Yaskawa INFORM job: aprem2TRJ0.JBI

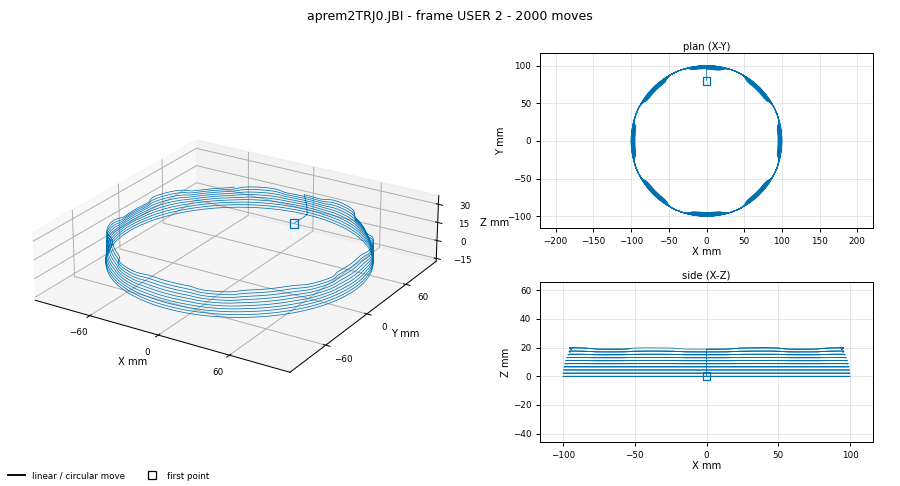
[picture p0: tool path of aprem2TRJ0.JBI in frame USER 2, 2000 of 2000 moves have a stored position in this frame; points joined in program order, loops and branches not executed]
/JOB
//NAME aprem2TRJ0
//POS
///NPOS 2000,0,2000,0,0,0
///USER 2
///TOOL 1
///POSTYPE USER
///RECTAN
///RCONF 1,0,0,0,0,0,0,0,0,0,0,0,0,0,0,0,0,0,0,0,0,0,0,0
C00000=0.000,80.000,0.000,-180.0000,0.0000,0.0000
C00001=0.000,100.000,0.000,-180.0000,0.0000,0.0000
C00002=5.792,99.832,0.000,-180.0000,-0.0000,0.0000
C00003=10.988,99.394,0.000,-180.0000,-0.0000,0.0000
C00004=15.564,98.781,0.000,-180.0000,-0.0000,0.0000
C00005=18.698,98.237,0.000,-180.0000,-0.0000,0.0000
C00006=20.854,97.801,0.000,-180.0000,-0.0000,0.0000
C00007=22.593,97.414,0.000,-180.0000,-0.0000,0.0000
C00008=24.351,96.990,0.000,-180.0000,-0.0000,0.0000
C00009=26.550,96.411,0.000,-180.0000,-0.0000,0.0000
C00010=29.248,95.627,0.000,-180.0000,-0.0000,0.0000
C00011=32.094,94.710,0.000,-180.0000,-0.0000,0.0000
C00012=34.739,93.772,0.000,-180.0000,-0.0000,0.0000
C00013=37.121,92.855,0.000,-180.0000,-0.0000,0.0000
C00014=39.410,91.907,0.000,-180.0000,-0.0000,0.0000
C00015=41.743,90.871,0.000,-180.0000,-0.0000,0.0000
C00016=44.276,89.664,0.000,180.0000,0.0000,0.0000
C00017=46.937,88.300,0.000,180.0000,0.0000,0.0000
C00018=49.400,86.946,0.000,-180.0000,-0.0000,0.0000
C00019=51.363,85.801,0.000,-180.0000,-0.0000,0.0000
C00020=52.906,84.858,0.000,-180.0000,-0.0000,0.0000
C00021=54.410,83.902,0.000,-180.0000,-0.0000,0.0000
C00022=56.242,82.685,0.000,-180.0000,-0.0000,0.0000
C00023=58.844,80.854,0.000,-180.0000,-0.0000,0.0000
C00024=62.512,78.053,0.000,-180.0000,-0.0000,0.0000
C00025=66.496,74.687,0.000,-180.0000,-0.0000,0.0000
C00026=70.711,70.711,0.000,-180.0000,-0.0000,0.0000
C00027=74.687,66.496,0.000,-180.0000,-0.0000,0.0000
C00028=78.053,62.512,0.000,-180.0000,-0.0000,0.0000
C00029=80.854,58.844,0.000,180.0000,0.0000,0.0000
C00030=82.685,56.242,0.000,-180.0000,-0.0000,0.0000
C00031=83.902,54.410,0.000,-180.0000,-0.0000,0.0000
C00032=84.858,52.906,0.000,-180.0000,-0.0000,0.0000
C00033=85.801,51.363,0.000,-180.0000,-0.0000,0.0000
C00034=86.946,49.400,0.000,-180.0000,-0.0000,0.0000
C00035=88.300,46.937,0.000,-180.0000,-0.0000,0.0000
C00036=89.664,44.276,0.000,-180.0000,-0.0000,0.0000
C00037=90.871,41.743,0.000,-180.0000,-0.0000,0.0000
C00038=91.907,39.410,0.000,-180.0000,-0.0000,0.0000
C00039=92.855,37.121,0.000,-180.0000,-0.0000,0.0000
C00040=93.772,34.739,0.000,-180.0000,-0.0000,0.0000
C00041=94.710,32.094,0.000,-180.0000,-0.0000,0.0000
C00042=95.627,29.248,0.000,-180.0000,-0.0000,0.0000
C00043=96.411,26.550,0.000,-180.0000,-0.0000,0.0000
C00044=96.990,24.351,0.000,-180.0000,-0.0000,0.0000
C00045=97.414,22.593,0.000,-180.0000,-0.0000,0.0000
C00046=97.801,20.854,0.000,-180.0000,-0.0000,0.0000
C00047=98.237,18.698,0.000,-180.0000,-0.0000,0.0000
C00048=98.781,15.564,0.000,-180.0000,-0.0000,0.0000
C00049=99.394,10.988,0.000,-180.0000,-0.0000,0.0000
C00050=99.832,5.792,0.000,-180.0000,-0.0000,0.0000
C00051=100.000,0.000,0.000,-180.0000,-0.0000,0.0000
C00052=99.832,-5.792,0.000,180.0000,-0.0000,0.0000
C00053=99.394,-10.988,0.000,180.0000,-0.0000,0.0000
C00054=98.781,-15.564,0.000,180.0000,-0.0000,0.0000
C00055=98.237,-18.698,0.000,180.0000,-0.0000,0.0000
C00056=97.801,-20.854,0.000,180.0000,-0.0000,0.0000
C00057=97.414,-22.593,0.000,180.0000,-0.0000,0.0000
C00058=96.990,-24.351,0.000,180.0000,-0.0000,0.0000
C00059=96.411,-26.550,0.000,180.0000,-0.0000,0.0000
C00060=95.627,-29.248,0.000,180.0000,-0.0000,0.0000
C00061=94.710,-32.094,0.000,180.0000,-0.0000,0.0000
C00062=93.772,-34.739,0.000,180.0000,-0.0000,0.0000
C00063=92.855,-37.121,0.000,180.0000,-0.0000,0.0000
C00064=91.907,-39.410,0.000,180.0000,-0.0000,0.0000
C00065=90.871,-41.743,0.000,180.0000,-0.0000,0.0000
C00066=89.664,-44.276,0.000,180.0000,-0.0000,0.0000
C00067=88.300,-46.937,0.000,180.0000,-0.0000,0.0000
C00068=86.946,-49.400,0.000,180.0000,-0.0000,0.0000
C00069=85.801,-51.363,0.000,180.0000,-0.0000,0.0000
C00070=84.858,-52.906,0.000,180.0000,-0.0000,0.0000
C00071=83.902,-54.410,0.000,180.0000,-0.0000,0.0000
C00072=82.685,-56.242,0.000,180.0000,-0.0000,0.0000
C00073=80.854,-58.844,0.000,180.0000,-0.0000,0.0000
C00074=78.053,-62.512,0.000,180.0000,-0.0000,0.0000
C00075=74.687,-66.496,0.000,180.0000,-0.0000,0.0000
C00076=70.711,-70.711,0.000,180.0000,-0.0000,0.0000
C00077=66.496,-74.687,0.000,180.0000,-0.0000,0.0000
C00078=62.512,-78.053,0.000,180.0000,-0.0000,0.0000
C00079=58.844,-80.854,0.000,180.0000,-0.0000,0.0000
C00080=56.242,-82.685,0.000,180.0000,-0.0000,0.0000
C00081=54.410,-83.902,0.000,180.0000,-0.0000,0.0000
C00082=52.906,-84.858,0.000,180.0000,-0.0000,0.0000
C00083=51.363,-85.801,0.000,180.0000,-0.0000,0.0000
C00084=49.400,-86.946,0.000,-180.0000,0.0000,0.0000
C00085=46.937,-88.300,0.000,180.0000,-0.0000,0.0000
C00086=44.276,-89.664,0.000,180.0000,-0.0000,0.0000
C00087=41.743,-90.871,0.000,180.0000,-0.0000,0.0000
C00088=39.410,-91.907,0.000,180.0000,-0.0000,0.0000
C00089=37.121,-92.855,0.000,180.0000,-0.0000,0.0000
C00090=34.739,-93.772,0.000,180.0000,-0.0000,0.0000
C00091=32.094,-94.710,0.000,180.0000,-0.0000,0.0000
C00092=29.248,-95.627,0.000,180.0000,-0.0000,0.0000
C00093=26.550,-96.411,0.000,180.0000,-0.0000,0.0000
C00094=24.351,-96.990,0.000,180.0000,-0.0000,0.0000
C00095=22.593,-97.414,0.000,180.0000,-0.0000,0.0000
C00096=20.854,-97.801,0.000,180.0000,-0.0000,0.0000
C00097=18.698,-98.237,0.000,180.0000,-0.0000,0.0000
C00098=15.564,-98.781,0.000,180.0000,-0.0000,0.0000
C00099=10.988,-99.394,0.000,180.0000,-0.0000,0.0000
C00100=5.792,-99.832,0.000,180.0000,-0.0000,0.0000
C00101=0.000,-100.000,0.000,-180.0000,-0.0000,0.0000
C00102=0.000,-100.000,0.000,-180.0000,-0.0000,0.0000
C00103=-5.792,-99.832,0.000,-180.0000,-0.0000,0.0000
C00104=-10.988,-99.394,0.000,-180.0000,-0.0000,0.0000
C00105=-15.564,-98.781,0.000,-180.0000,-0.0000,0.0000
C00106=-18.698,-98.237,0.000,-180.0000,-0.0000,0.0000
C00107=-20.854,-97.801,0.000,-180.0000,-0.0000,0.0000
C00108=-22.593,-97.414,0.000,-180.0000,-0.0000,0.0000
C00109=-24.351,-96.990,0.000,-180.0000,-0.0000,0.0000
C00110=-26.550,-96.411,0.000,-180.0000,-0.0000,0.0000
C00111=-29.248,-95.627,0.000,-180.0000,-0.0000,0.0000
C00112=-32.094,-94.710,0.000,-180.0000,-0.0000,0.0000
C00113=-34.739,-93.772,0.000,-180.0000,-0.0000,0.0000
C00114=-37.121,-92.855,0.000,-180.0000,-0.0000,0.0000
C00115=-39.410,-91.907,0.000,-180.0000,-0.0000,0.0000
C00116=-41.743,-90.871,0.000,-180.0000,-0.0000,0.0000
C00117=-44.276,-89.664,0.000,-180.0000,-0.0000,0.0000
C00118=-46.937,-88.300,0.000,-180.0000,-0.0000,0.0000
C00119=-49.400,-86.946,0.000,-180.0000,-0.0000,0.0000
C00120=-51.363,-85.801,0.000,-180.0000,-0.0000,0.0000
C00121=-52.906,-84.858,0.000,-180.0000,-0.0000,0.0000
C00122=-54.410,-83.902,0.000,-180.0000,-0.0000,0.0000
C00123=-56.242,-82.685,0.000,-180.0000,-0.0000,0.0000
C00124=-58.844,-80.854,0.000,-180.0000,-0.0000,0.0000
C00125=-62.512,-78.053,0.000,-180.0000,-0.0000,0.0000
C00126=-66.496,-74.687,0.000,-180.0000,-0.0000,0.0000
C00127=-70.711,-70.711,0.000,-180.0000,-0.0000,0.0000
C00128=-74.687,-66.496,0.000,-180.0000,-0.0000,0.0000
C00129=-78.053,-62.512,0.000,-180.0000,-0.0000,0.0000
C00130=-80.854,-58.844,0.000,-180.0000,-0.0000,0.0000
C00131=-82.685,-56.242,0.000,-180.0000,-0.0000,0.0000
C00132=-83.902,-54.410,0.000,-180.0000,-0.0000,0.0000
C00133=-84.858,-52.906,0.000,-180.0000,-0.0000,0.0000
C00134=-85.801,-51.363,0.000,-180.0000,-0.0000,0.0000
C00135=-86.946,-49.400,0.000,-180.0000,-0.0000,0.0000
C00136=-88.300,-46.937,0.000,-180.0000,-0.0000,0.0000
C00137=-89.664,-44.276,0.000,-180.0000,-0.0000,0.0000
C00138=-90.871,-41.743,0.000,180.0000,0.0000,0.0000
C00139=-91.907,-39.410,0.000,180.0000,0.0000,0.0000
C00140=-92.855,-37.121,0.000,-180.0000,-0.0000,0.0000
C00141=-93.772,-34.739,0.000,-180.0000,-0.0000,0.0000
C00142=-94.710,-32.094,0.000,180.0000,0.0000,0.0000
C00143=-95.627,-29.248,0.000,180.0000,0.0000,0.0000
C00144=-96.411,-26.550,0.000,-180.0000,-0.0000,0.0000
C00145=-96.990,-24.351,0.000,-180.0000,-0.0000,0.0000
C00146=-97.414,-22.593,0.000,-180.0000,-0.0000,0.0000
C00147=-97.801,-20.854,0.000,-180.0000,-0.0000,0.0000
C00148=-98.237,-18.698,0.000,-180.0000,-0.0000,0.0000
C00149=-98.781,-15.564,0.000,-180.0000,-0.0000,0.0000
C00150=-99.394,-10.988,0.000,-180.0000,-0.0000,0.0000
C00151=-99.832,-5.792,0.000,-180.0000,-0.0000,0.0000
C00152=-100.000,0.000,0.000,180.0000,0.0000,0.0000
C00153=-99.832,5.792,0.000,-180.0000,0.0000,0.0000
C00154=-99.394,10.988,0.000,-180.0000,0.0000,0.0000
C00155=-98.781,15.564,0.000,-180.0000,0.0000,0.0000
C00156=-98.237,18.698,0.000,-180.0000,0.0000,0.0000
C00157=-97.801,20.854,0.000,-180.0000,0.0000,0.0000
C00158=-97.414,22.593,0.000,-180.0000,0.0000,0.0000
C00159=-96.990,24.351,0.000,-180.0000,0.0000,0.0000
C00160=-96.411,26.550,0.000,-180.0000,0.0000,0.0000
C00161=-95.627,29.248,0.000,-180.0000,0.0000,0.0000
C00162=-94.710,32.094,0.000,-180.0000,0.0000,0.0000
C00163=-93.772,34.739,0.000,-180.0000,0.0000,0.0000
C00164=-92.855,37.121,0.000,-180.0000,0.0000,0.0000
C00165=-91.907,39.410,0.000,-180.0000,0.0000,0.0000
C00166=-90.871,41.743,0.000,-180.0000,0.0000,0.0000
C00167=-89.664,44.276,0.000,-180.0000,0.0000,0.0000
C00168=-88.300,46.937,0.000,-180.0000,0.0000,0.0000
C00169=-86.946,49.400,0.000,-180.0000,0.0000,0.0000
C00170=-85.801,51.363,0.000,-180.0000,0.0000,0.0000
C00171=-84.858,52.906,0.000,-180.0000,0.0000,0.0000
C00172=-83.902,54.410,0.000,-180.0000,0.0000,0.0000
C00173=-82.685,56.242,0.000,-180.0000,0.0000,0.0000
C00174=-80.854,58.844,0.000,-180.0000,0.0000,0.0000
C00175=-78.053,62.512,0.000,-180.0000,0.0000,0.0000
C00176=-74.687,66.496,0.000,-180.0000,0.0000,0.0000
C00177=-70.711,70.711,0.000,-180.0000,0.0000,0.0000
C00178=-66.496,74.687,0.000,-180.0000,0.0000,0.0000
C00179=-62.512,78.053,0.000,-180.0000,0.0000,0.0000
C00180=-58.844,80.854,0.000,-180.0000,0.0000,0.0000
C00181=-56.242,82.685,0.000,-180.0000,0.0000,0.0000
C00182=-54.410,83.902,0.000,-180.0000,0.0000,0.0000
C00183=-52.906,84.858,0.000,-180.0000,0.0000,0.0000
C00184=-51.363,85.801,0.000,-180.0000,0.0000,0.0000
C00185=-49.400,86.946,0.000,-180.0000,0.0000,0.0000
C00186=-46.937,88.300,0.000,-180.0000,0.0000,0.0000
C00187=-44.276,89.664,0.000,-180.0000,0.0000,0.0000
C00188=-41.743,90.871,0.000,-180.0000,0.0000,0.0000
C00189=-39.410,91.907,0.000,-180.0000,0.0000,0.0000
C00190=-37.121,92.855,0.000,-180.0000,0.0000,0.0000
C00191=-34.739,93.772,0.000,-180.0000,0.0000,0.0000
C00192=-32.094,94.710,0.000,-180.0000,0.0000,0.0000
C00193=-29.248,95.627,0.000,-180.0000,0.0000,0.0000
C00194=-26.550,96.411,0.000,-180.0000,0.0000,0.0000
C00195=-24.351,96.990,0.000,-180.0000,0.0000,0.0000
C00196=-22.593,97.414,0.000,-180.0000,0.0000,0.0000
C00197=-20.854,97.801,0.000,-180.0000,0.0000,0.0000
C00198=-18.698,98.237,0.000,-180.0000,0.0000,0.0000
C00199=-15.564,98.781,0.000,-180.0000,0.0000,0.0000
C00200=-10.988,99.394,0.000,-180.0000,0.0000,0.0000
C00201=-5.792,99.832,0.000,-180.0000,0.0000,0.0000
C00202=0.000,100.000,0.000,-180.0000,0.0000,0.0000
C00203=0.000,99.921,2.199,-175.9398,0.0000,0.0000
C00204=5.785,99.754,2.199,-175.9444,-0.2364,0.0000
C00205=10.976,99.317,2.199,-175.9703,-0.4452,0.0000
C00206=15.549,98.707,2.199,-176.1463,-0.6026,0.0000
C00207=18.681,98.171,2.199,-176.5600,-0.6415,0.0000
C00208=20.835,97.748,2.199,-177.1484,-0.5884,0.0000
C00209=22.573,97.375,2.200,-177.8314,-0.4845,0.0000
C00210=24.330,96.965,2.200,-178.5159,-0.3619,0.0000
C00211=26.527,96.399,2.200,-179.1045,-0.2425,0.0000
C00212=29.226,95.625,2.200,-179.5721,-0.1295,0.0000
C00213=32.077,94.713,2.200,-179.8787,-0.0409,0.0000
C00214=34.728,93.776,2.200,-179.9807,-0.0071,0.0000
C00215=37.118,92.856,2.200,-179.9977,-0.0009,0.0000
C00216=39.413,91.905,2.200,-179.9978,-0.0010,0.0000
C00217=41.753,90.866,2.200,-179.9813,-0.0086,0.0000
C00218=44.291,89.654,2.200,-179.8853,-0.0569,0.0000
C00219=46.951,88.283,2.200,-179.6059,-0.2110,0.0000
C00220=49.407,86.922,2.200,-179.1953,-0.4618,0.0000
C00221=51.360,85.768,2.200,-178.6947,-0.7937,0.0000
C00222=52.893,84.816,2.200,-178.1239,-1.1914,0.0000
C00223=54.385,83.851,2.199,-177.5673,-1.6016,0.0000
C00224=56.208,82.627,2.199,-177.1135,-1.9809,0.0000
C00225=58.802,80.791,2.199,-176.8480,-2.3017,0.0000
C00226=62.466,77.989,2.199,-176.8343,-2.5377,0.0000
C00227=66.446,74.627,2.199,-176.9631,-2.7034,0.0000
C00228=70.655,70.655,2.199,-177.1266,-2.8734,0.0000
C00229=74.627,66.446,2.199,-177.2966,-3.0369,0.0000
C00230=77.989,62.466,2.199,-177.4623,-3.1657,0.0000
C00231=80.791,58.802,2.199,-177.6983,-3.1520,0.0000
C00232=82.627,56.208,2.199,-178.0191,-2.8865,0.0000
C00233=83.851,54.385,2.199,-178.3984,-2.4327,0.0000
C00234=84.816,52.893,2.200,-178.8086,-1.8761,0.0000
C00235=85.768,51.360,2.200,-179.2063,-1.3053,0.0000
C00236=86.922,49.407,2.200,-179.5382,-0.8047,0.0000
C00237=88.283,46.951,2.200,-179.7890,-0.3941,0.0000
C00238=89.654,44.291,2.200,-179.9431,-0.1147,0.0000
C00239=90.866,41.753,2.200,-179.9914,-0.0187,0.0000
C00240=91.905,39.413,2.200,-179.9990,-0.0022,0.0000
C00241=92.856,37.118,2.200,-179.9991,-0.0023,0.0000
C00242=93.776,34.728,2.200,-179.9929,-0.0193,0.0000
C00243=94.713,32.077,2.200,-179.9591,-0.1213,0.0000
C00244=95.625,29.226,2.200,-179.8705,-0.4279,0.0000
C00245=96.399,26.527,2.200,-179.7575,-0.8955,0.0000
C00246=96.965,24.330,2.200,-179.6381,-1.4841,0.0000
C00247=97.375,22.573,2.200,-179.5155,-2.1686,0.0000
C00248=97.748,20.835,2.199,-179.4116,-2.8516,0.0000
C00249=98.171,18.681,2.199,-179.3585,-3.4400,0.0000
C00250=98.707,15.549,2.199,-179.3974,-3.8537,0.0000
C00251=99.317,10.976,2.199,-179.5548,-4.0297,0.0000
C00252=99.754,5.785,2.199,-179.7636,-4.0556,0.0000
C00253=99.921,0.000,2.199,180.0000,-4.0602,0.0000
C00254=99.754,-5.785,2.199,179.7636,-4.0556,0.0000
C00255=99.317,-10.976,2.199,179.5548,-4.0297,0.0000
C00256=98.707,-15.549,2.199,179.3974,-3.8537,0.0000
C00257=98.171,-18.681,2.199,179.3585,-3.4400,0.0000
C00258=97.748,-20.835,2.199,179.4116,-2.8516,0.0000
C00259=97.375,-22.573,2.200,179.5155,-2.1686,0.0000
C00260=96.965,-24.330,2.200,179.6381,-1.4841,0.0000
C00261=96.399,-26.527,2.200,179.7575,-0.8955,0.0000
C00262=95.625,-29.226,2.200,179.8705,-0.4279,0.0000
C00263=94.713,-32.077,2.200,179.9591,-0.1213,0.0000
C00264=93.776,-34.728,2.200,179.9929,-0.0193,0.0000
C00265=92.856,-37.118,2.200,179.9991,-0.0023,0.0000
C00266=91.905,-39.413,2.200,179.9990,-0.0022,0.0000
C00267=90.866,-41.753,2.200,179.9914,-0.0187,0.0000
C00268=89.654,-44.291,2.200,179.9431,-0.1147,0.0000
C00269=88.283,-46.951,2.200,179.7890,-0.3941,0.0000
C00270=86.922,-49.407,2.200,179.5382,-0.8047,0.0000
C00271=85.768,-51.360,2.200,179.2063,-1.3053,0.0000
C00272=84.816,-52.893,2.200,178.8086,-1.8761,0.0000
C00273=83.851,-54.385,2.199,178.3984,-2.4327,0.0000
C00274=82.627,-56.208,2.199,178.0191,-2.8865,0.0000
C00275=80.791,-58.802,2.199,177.6983,-3.1520,0.0000
C00276=77.989,-62.466,2.199,177.4623,-3.1657,0.0000
C00277=74.627,-66.446,2.199,177.2966,-3.0369,0.0000
C00278=70.655,-70.655,2.199,177.1266,-2.8734,0.0000
C00279=66.446,-74.627,2.199,176.9631,-2.7034,0.0000
C00280=62.466,-77.989,2.199,176.8343,-2.5377,0.0000
C00281=58.802,-80.791,2.199,176.8480,-2.3017,0.0000
C00282=56.208,-82.627,2.199,177.1135,-1.9809,0.0000
C00283=54.385,-83.851,2.199,177.5673,-1.6016,0.0000
C00284=52.893,-84.816,2.200,178.1239,-1.1914,0.0000
C00285=51.360,-85.768,2.200,178.6947,-0.7937,0.0000
C00286=49.407,-86.922,2.200,179.1953,-0.4618,0.0000
C00287=46.951,-88.283,2.200,179.6059,-0.2110,0.0000
C00288=44.291,-89.654,2.200,179.8853,-0.0569,0.0000
C00289=41.753,-90.866,2.200,179.9813,-0.0086,0.0000
C00290=39.413,-91.905,2.200,179.9978,-0.0010,0.0000
C00291=37.118,-92.856,2.200,179.9977,-0.0009,0.0000
C00292=34.728,-93.776,2.200,179.9807,-0.0071,0.0000
C00293=32.077,-94.713,2.200,179.8787,-0.0409,0.0000
C00294=29.226,-95.625,2.200,179.5721,-0.1295,0.0000
C00295=26.527,-96.399,2.200,179.1045,-0.2425,0.0000
C00296=24.330,-96.965,2.200,178.5159,-0.3619,0.0000
C00297=22.573,-97.375,2.200,177.8314,-0.4845,0.0000
C00298=20.835,-97.748,2.199,177.1484,-0.5884,0.0000
C00299=18.681,-98.171,2.199,176.5600,-0.6415,0.0000
C00300=15.549,-98.707,2.199,176.1463,-0.6026,0.0000
C00301=10.976,-99.317,2.199,175.9703,-0.4452,0.0000
C00302=5.785,-99.754,2.199,175.9444,-0.2364,0.0000
C00303=0.000,-99.921,2.199,175.9398,0.0000,0.0000
C00304=0.000,-99.921,2.199,175.9398,0.0000,0.0000
C00305=-5.785,-99.754,2.199,175.9444,0.2364,0.0000
C00306=-10.976,-99.317,2.199,175.9703,0.4452,0.0000
C00307=-15.549,-98.707,2.199,176.1463,0.6026,0.0000
C00308=-18.681,-98.171,2.199,176.5600,0.6415,0.0000
C00309=-20.835,-97.748,2.199,177.1484,0.5884,0.0000
C00310=-22.573,-97.375,2.200,177.8314,0.4845,0.0000
C00311=-24.330,-96.965,2.200,178.5159,0.3619,0.0000
C00312=-26.527,-96.399,2.200,179.1045,0.2425,0.0000
C00313=-29.226,-95.625,2.200,179.5721,0.1295,0.0000
C00314=-32.077,-94.713,2.200,179.8787,0.0409,0.0000
C00315=-34.728,-93.776,2.200,179.9807,0.0071,0.0000
C00316=-37.118,-92.856,2.200,179.9977,0.0009,0.0000
C00317=-39.413,-91.905,2.200,179.9978,0.0010,0.0000
C00318=-41.753,-90.866,2.200,179.9813,0.0086,0.0000
C00319=-44.291,-89.654,2.200,179.8853,0.0569,0.0000
C00320=-46.951,-88.283,2.200,179.6059,0.2110,0.0000
C00321=-49.407,-86.922,2.200,179.1953,0.4618,0.0000
C00322=-51.360,-85.768,2.200,178.6947,0.7937,0.0000
C00323=-52.893,-84.816,2.200,178.1239,1.1914,0.0000
C00324=-54.385,-83.851,2.199,177.5673,1.6016,0.0000
C00325=-56.208,-82.627,2.199,177.1135,1.9809,0.0000
C00326=-58.802,-80.791,2.199,176.8480,2.3017,0.0000
C00327=-62.466,-77.989,2.199,176.8343,2.5377,0.0000
C00328=-66.446,-74.627,2.199,176.9631,2.7034,0.0000
C00329=-70.655,-70.655,2.199,177.1266,2.8734,0.0000
C00330=-74.627,-66.446,2.199,177.2966,3.0369,0.0000
C00331=-77.989,-62.466,2.199,177.4623,3.1657,0.0000
C00332=-80.791,-58.802,2.199,177.6983,3.1520,0.0000
C00333=-82.627,-56.208,2.199,178.0191,2.8865,0.0000
C00334=-83.851,-54.385,2.199,178.3984,2.4327,0.0000
C00335=-84.816,-52.893,2.200,178.8086,1.8761,0.0000
C00336=-85.768,-51.360,2.200,179.2063,1.3053,0.0000
C00337=-86.922,-49.407,2.200,179.5382,0.8047,0.0000
C00338=-88.283,-46.951,2.200,179.7890,0.3941,0.0000
C00339=-89.654,-44.291,2.200,179.9431,0.1147,0.0000
C00340=-90.866,-41.753,2.200,179.9914,0.0187,0.0000
C00341=-91.905,-39.413,2.200,179.9990,0.0022,0.0000
C00342=-92.856,-37.118,2.200,179.9991,0.0023,0.0000
C00343=-93.776,-34.728,2.200,179.9929,0.0193,0.0000
C00344=-94.713,-32.077,2.200,179.9591,0.1213,0.0000
C00345=-95.625,-29.226,2.200,179.8705,0.4279,0.0000
C00346=-96.399,-26.527,2.200,179.7575,0.8955,0.0000
C00347=-96.965,-24.330,2.200,179.6381,1.4841,0.0000
C00348=-97.375,-22.573,2.200,179.5155,2.1686,0.0000
C00349=-97.748,-20.835,2.199,179.4116,2.8516,0.0000
C00350=-98.171,-18.681,2.199,179.3585,3.4400,0.0000
C00351=-98.707,-15.549,2.199,179.3974,3.8537,0.0000
C00352=-99.317,-10.976,2.199,179.5548,4.0297,0.0000
C00353=-99.754,-5.785,2.199,179.7636,4.0556,0.0000
C00354=-99.921,0.000,2.199,-180.0000,4.0602,0.0000
C00355=-99.754,5.785,2.199,-179.7636,4.0556,0.0000
C00356=-99.317,10.976,2.199,-179.5548,4.0297,0.0000
C00357=-98.707,15.549,2.199,-179.3974,3.8537,0.0000
C00358=-98.171,18.681,2.199,-179.3585,3.4400,0.0000
C00359=-97.748,20.835,2.199,-179.4116,2.8516,0.0000
C00360=-97.375,22.573,2.200,-179.5155,2.1686,0.0000
C00361=-96.965,24.330,2.200,-179.6381,1.4841,0.0000
C00362=-96.399,26.527,2.200,-179.7575,0.8955,0.0000
C00363=-95.625,29.226,2.200,-179.8705,0.4279,0.0000
C00364=-94.713,32.077,2.200,-179.9591,0.1213,0.0000
C00365=-93.776,34.728,2.200,-179.9929,0.0193,0.0000
C00366=-92.856,37.118,2.200,-179.9991,0.0023,0.0000
C00367=-91.905,39.413,2.200,-179.9990,0.0022,0.0000
C00368=-90.866,41.753,2.200,-179.9914,0.0187,0.0000
C00369=-89.654,44.291,2.200,-179.9431,0.1147,0.0000
C00370=-88.283,46.951,2.200,-179.7890,0.3941,0.0000
C00371=-86.922,49.407,2.200,-179.5382,0.8047,0.0000
C00372=-85.768,51.360,2.200,-179.2063,1.3053,0.0000
C00373=-84.816,52.893,2.200,-178.8086,1.8761,0.0000
C00374=-83.851,54.385,2.199,-178.3984,2.4327,0.0000
C00375=-82.627,56.208,2.199,-178.0191,2.8865,0.0000
C00376=-80.791,58.802,2.199,-177.6983,3.1520,0.0000
C00377=-77.989,62.466,2.199,-177.4623,3.1657,0.0000
C00378=-74.627,66.446,2.199,-177.2966,3.0369,0.0000
C00379=-70.655,70.655,2.199,-177.1266,2.8734,0.0000
C00380=-66.446,74.627,2.199,-176.9631,2.7034,0.0000
C00381=-62.466,77.989,2.199,-176.8343,2.5377,0.0000
C00382=-58.802,80.791,2.199,-176.8480,2.3017,0.0000
C00383=-56.208,82.627,2.199,-177.1135,1.9809,0.0000
C00384=-54.385,83.851,2.199,-177.5673,1.6016,0.0000
C00385=-52.893,84.816,2.200,-178.1239,1.1914,0.0000
C00386=-51.360,85.768,2.200,-178.6947,0.7937,0.0000
C00387=-49.407,86.922,2.200,-179.1953,0.4618,0.0000
C00388=-46.951,88.283,2.200,-179.6059,0.2110,0.0000
C00389=-44.291,89.654,2.200,-179.8853,0.0569,0.0000
C00390=-41.753,90.866,2.200,-179.9813,0.0086,0.0000
C00391=-39.413,91.905,2.200,-179.9978,0.0010,0.0000
C00392=-37.118,92.856,2.200,-179.9977,0.0009,0.0000
C00393=-34.728,93.776,2.200,-179.9807,0.0071,0.0000
C00394=-32.077,94.713,2.200,-179.8787,0.0409,0.0000
C00395=-29.226,95.625,2.200,-179.5721,0.1295,0.0000
C00396=-26.527,96.399,2.200,-179.1045,0.2425,0.0000
C00397=-24.330,96.965,2.200,-178.5159,0.3619,0.0000
C00398=-22.573,97.375,2.200,-177.8314,0.4845,0.0000
C00399=-20.835,97.748,2.199,-177.1484,0.5884,0.0000
C00400=-18.681,98.171,2.199,-176.5600,0.6415,0.0000
C00401=-15.549,98.707,2.199,-176.1463,0.6026,0.0000
C00402=-10.976,99.317,2.199,-175.9703,0.4452,0.0000
C00403=-5.785,99.754,2.199,-175.9444,0.2364,0.0000
C00404=0.000,99.921,2.199,-175.9398,0.0000,0.0000
C00405=0.000,99.691,4.387,-172.1026,0.0000,0.0000
C00406=5.764,99.524,4.387,-172.1115,-0.4617,0.0000
C00407=10.941,99.090,4.387,-172.1612,-0.8645,0.0000
C00408=15.506,98.490,4.388,-172.4978,-1.1464,0.0000
C00409=18.630,97.979,4.390,-173.2935,-1.1748,0.0000
C00410=20.779,97.591,4.393,-174.4370,-1.0358,0.0000
C00411=22.514,97.259,4.396,-175.7755,-0.8390,0.0000
C00412=24.268,96.890,4.398,-177.1185,-0.6429,0.0000
C00413=26.460,96.362,4.399,-178.2686,-0.4458,0.0000
C00414=29.164,95.617,4.399,-179.1783,-0.2412,0.0000
C00415=32.027,94.722,4.399,-179.7705,-0.0761,0.0000
C00416=34.697,93.786,4.400,-179.9632,-0.0136,0.0000
C00417=37.107,92.860,4.400,-179.9957,-0.0017,0.0000
C00418=39.424,91.901,4.400,-179.9957,-0.0018,0.0000
C00419=41.782,90.851,4.400,-179.9644,-0.0164,0.0000
C00420=44.332,89.625,4.399,-179.7839,-0.1085,0.0000
C00421=46.990,88.233,4.399,-179.2484,-0.4105,0.0000
C00422=49.428,86.848,4.399,-178.4605,-0.9093,0.0000
C00423=51.352,85.672,4.398,-177.5077,-1.5842,0.0000
C00424=52.853,84.692,4.396,-176.4188,-2.3979,0.0000
C00425=54.314,83.700,4.393,-175.3318,-3.2102,0.0000
C00426=56.108,82.455,4.390,-174.4229,-3.9270,0.0000
C00427=58.679,80.608,4.388,-173.8773,-4.5153,0.0000
C00428=62.331,77.804,4.387,-173.8348,-4.9540,0.0000
C00429=66.299,74.450,4.387,-174.0811,-5.2722,0.0000
C00430=70.493,70.493,4.387,-174.3980,-5.6020,0.0000
C00431=74.450,66.299,4.387,-174.7278,-5.9188,0.0000
C00432=77.804,62.331,4.387,-175.0460,-6.1652,0.0000
C00433=80.608,58.679,4.388,-175.4847,-6.1227,0.0000
C00434=82.455,56.108,4.390,-176.0730,-5.5771,0.0000
C00435=83.700,54.314,4.393,-176.7898,-4.6682,0.0000
C00436=84.692,52.853,4.396,-177.6021,-3.5812,0.0000
C00437=85.672,51.352,4.398,-178.4158,-2.4923,0.0000
C00438=86.848,49.428,4.399,-179.0907,-1.5395,0.0000
C00439=88.233,46.990,4.399,-179.5895,-0.7516,0.0000
C00440=89.625,44.332,4.399,-179.8915,-0.2161,0.0000
C00441=90.851,41.782,4.400,-179.9836,-0.0356,0.0000
C00442=91.901,39.424,4.400,-179.9982,-0.0043,0.0000
C00443=92.860,37.107,4.400,-179.9983,-0.0043,0.0000
C00444=93.786,34.697,4.400,-179.9864,-0.0368,0.0000
C00445=94.722,32.027,4.399,-179.9239,-0.2295,0.0000
C00446=95.617,29.164,4.399,-179.7588,-0.8217,0.0000
C00447=96.362,26.460,4.399,-179.5542,-1.7314,0.0000
C00448=96.890,24.268,4.398,-179.3571,-2.8815,0.0000
C00449=97.259,22.514,4.396,-179.1610,-4.2245,0.0000
C00450=97.591,20.779,4.393,-178.9642,-5.5630,0.0000
C00451=97.979,18.630,4.390,-178.8252,-6.7065,0.0000
C00452=98.490,15.506,4.388,-178.8536,-7.5022,0.0000
C00453=99.090,10.941,4.387,-179.1355,-7.8388,0.0000
C00454=99.524,5.764,4.387,-179.5383,-7.8885,0.0000
C00455=99.691,0.000,4.387,180.0000,-7.8974,0.0000
C00456=99.524,-5.764,4.387,179.5383,-7.8885,0.0000
C00457=99.090,-10.941,4.387,179.1355,-7.8388,0.0000
C00458=98.490,-15.506,4.388,178.8536,-7.5022,0.0000
C00459=97.979,-18.630,4.390,178.8252,-6.7065,0.0000
C00460=97.591,-20.779,4.393,178.9642,-5.5630,0.0000
C00461=97.259,-22.514,4.396,179.1610,-4.2245,0.0000
C00462=96.890,-24.268,4.398,179.3571,-2.8815,0.0000
C00463=96.362,-26.460,4.399,179.5542,-1.7314,0.0000
C00464=95.617,-29.164,4.399,179.7588,-0.8217,0.0000
C00465=94.722,-32.027,4.399,179.9239,-0.2295,0.0000
C00466=93.786,-34.697,4.400,179.9864,-0.0368,0.0000
C00467=92.860,-37.107,4.400,179.9983,-0.0043,0.0000
C00468=91.901,-39.424,4.400,179.9982,-0.0043,0.0000
C00469=90.851,-41.782,4.400,179.9836,-0.0356,0.0000
C00470=89.625,-44.332,4.399,179.8915,-0.2161,0.0000
C00471=88.233,-46.990,4.399,179.5895,-0.7516,0.0000
C00472=86.848,-49.428,4.399,179.0907,-1.5395,0.0000
C00473=85.672,-51.352,4.398,178.4158,-2.4923,0.0000
C00474=84.692,-52.853,4.396,177.6021,-3.5812,0.0000
C00475=83.700,-54.314,4.393,176.7898,-4.6682,0.0000
C00476=82.455,-56.108,4.390,176.0730,-5.5771,0.0000
C00477=80.608,-58.679,4.388,175.4847,-6.1227,0.0000
C00478=77.804,-62.331,4.387,175.0460,-6.1652,0.0000
C00479=74.450,-66.299,4.387,174.7278,-5.9189,0.0000
C00480=70.493,-70.493,4.387,174.3980,-5.6020,0.0000
C00481=66.299,-74.450,4.387,174.0812,-5.2722,0.0000
C00482=62.331,-77.804,4.387,173.8348,-4.9540,0.0000
C00483=58.679,-80.608,4.388,173.8773,-4.5153,0.0000
C00484=56.108,-82.455,4.390,174.4229,-3.9270,0.0000
C00485=54.314,-83.700,4.393,175.3318,-3.2102,0.0000
C00486=52.853,-84.692,4.396,176.4188,-2.3979,0.0000
C00487=51.352,-85.672,4.398,177.5077,-1.5842,0.0000
C00488=49.428,-86.848,4.399,178.4605,-0.9093,0.0000
C00489=46.990,-88.233,4.399,179.2484,-0.4105,0.0000
C00490=44.332,-89.625,4.399,179.7839,-0.1085,0.0000
C00491=41.782,-90.851,4.400,179.9644,-0.0164,0.0000
C00492=39.424,-91.901,4.400,179.9957,-0.0018,0.0000
C00493=37.107,-92.860,4.400,179.9957,-0.0017,0.0000
C00494=34.697,-93.786,4.400,179.9632,-0.0136,0.0000
C00495=32.027,-94.722,4.399,179.7705,-0.0761,0.0000
C00496=29.164,-95.617,4.399,179.1783,-0.2412,0.0000
C00497=26.460,-96.362,4.399,178.2686,-0.4458,0.0000
C00498=24.268,-96.890,4.398,177.1185,-0.6429,0.0000
C00499=22.514,-97.259,4.396,175.7755,-0.8390,0.0000
C00500=20.779,-97.591,4.393,174.4370,-1.0358,0.0000
C00501=18.630,-97.979,4.390,173.2935,-1.1748,0.0000
C00502=15.506,-98.490,4.388,172.4978,-1.1464,0.0000
C00503=10.941,-99.090,4.387,172.1612,-0.8645,0.0000
C00504=5.764,-99.524,4.387,172.1115,-0.4617,0.0000
C00505=0.000,-99.691,4.387,172.1026,0.0000,0.0000
C00506=0.000,-99.691,4.387,172.1026,0.0000,0.0000
C00507=-5.764,-99.524,4.387,172.1115,0.4617,0.0000
C00508=-10.941,-99.090,4.387,172.1612,0.8645,0.0000
C00509=-15.506,-98.490,4.388,172.4978,1.1464,0.0000
C00510=-18.630,-97.979,4.390,173.2935,1.1748,0.0000
C00511=-20.779,-97.591,4.393,174.4370,1.0358,0.0000
C00512=-22.514,-97.259,4.396,175.7755,0.8390,0.0000
C00513=-24.268,-96.890,4.398,177.1185,0.6429,0.0000
C00514=-26.460,-96.362,4.399,178.2686,0.4458,0.0000
C00515=-29.164,-95.617,4.399,179.1783,0.2412,0.0000
C00516=-32.027,-94.722,4.399,179.7705,0.0761,0.0000
C00517=-34.697,-93.786,4.400,179.9632,0.0136,0.0000
C00518=-37.107,-92.860,4.400,179.9957,0.0017,0.0000
C00519=-39.424,-91.901,4.400,179.9957,0.0018,0.0000
C00520=-41.782,-90.851,4.400,179.9644,0.0164,0.0000
C00521=-44.332,-89.625,4.399,179.7839,0.1085,0.0000
C00522=-46.990,-88.233,4.399,179.2484,0.4105,0.0000
C00523=-49.428,-86.848,4.399,178.4605,0.9093,0.0000
C00524=-51.352,-85.672,4.398,177.5077,1.5842,0.0000
C00525=-52.853,-84.692,4.396,176.4188,2.3979,0.0000
C00526=-54.314,-83.700,4.393,175.3318,3.2102,0.0000
C00527=-56.108,-82.455,4.390,174.4229,3.9270,0.0000
C00528=-58.679,-80.608,4.388,173.8773,4.5153,0.0000
C00529=-62.331,-77.804,4.387,173.8348,4.9540,0.0000
C00530=-66.299,-74.450,4.387,174.0811,5.2722,0.0000
C00531=-70.493,-70.493,4.387,174.3980,5.6020,0.0000
C00532=-74.450,-66.299,4.387,174.7278,5.9188,0.0000
C00533=-77.804,-62.331,4.387,175.0460,6.1652,0.0000
C00534=-80.608,-58.679,4.388,175.4847,6.1227,0.0000
C00535=-82.455,-56.108,4.390,176.0730,5.5771,0.0000
C00536=-83.700,-54.314,4.393,176.7898,4.6682,0.0000
C00537=-84.692,-52.853,4.396,177.6021,3.5812,0.0000
C00538=-85.672,-51.352,4.398,178.4158,2.4923,0.0000
C00539=-86.848,-49.428,4.399,179.0907,1.5395,0.0000
C00540=-88.233,-46.990,4.399,179.5895,0.7516,0.0000
C00541=-89.625,-44.332,4.399,179.8915,0.2161,0.0000
C00542=-90.851,-41.782,4.400,179.9836,0.0356,0.0000
C00543=-91.901,-39.424,4.400,179.9982,0.0043,0.0000
C00544=-92.860,-37.107,4.400,179.9983,0.0043,0.0000
C00545=-93.786,-34.697,4.400,179.9864,0.0368,0.0000
C00546=-94.722,-32.027,4.399,179.9239,0.2295,0.0000
C00547=-95.617,-29.164,4.399,179.7588,0.8217,0.0000
C00548=-96.362,-26.460,4.399,179.5542,1.7314,0.0000
C00549=-96.890,-24.268,4.398,179.3571,2.8815,0.0000
C00550=-97.259,-22.514,4.396,179.1610,4.2245,0.0000
C00551=-97.591,-20.779,4.393,178.9642,5.5630,0.0000
C00552=-97.979,-18.630,4.390,178.8252,6.7065,0.0000
C00553=-98.490,-15.506,4.388,178.8536,7.5022,0.0000
C00554=-99.090,-10.941,4.387,179.1355,7.8388,0.0000
C00555=-99.524,-5.764,4.387,179.5383,7.8885,0.0000
C00556=-99.691,0.000,4.387,-180.0000,7.8974,0.0000
C00557=-99.524,5.764,4.387,-179.5383,7.8885,0.0000
C00558=-99.090,10.941,4.387,-179.1355,7.8388,0.0000
C00559=-98.490,15.506,4.388,-178.8536,7.5022,0.0000
C00560=-97.979,18.630,4.390,-178.8252,6.7065,0.0000
C00561=-97.591,20.779,4.393,-178.9642,5.5630,0.0000
C00562=-97.259,22.514,4.396,-179.1610,4.2245,0.0000
C00563=-96.890,24.268,4.398,-179.3571,2.8815,0.0000
C00564=-96.362,26.460,4.399,-179.5542,1.7314,0.0000
C00565=-95.617,29.164,4.399,-179.7588,0.8217,0.0000
C00566=-94.722,32.027,4.399,-179.9239,0.2295,0.0000
C00567=-93.786,34.697,4.400,-179.9864,0.0368,0.0000
C00568=-92.860,37.107,4.400,-179.9983,0.0043,0.0000
C00569=-91.901,39.424,4.400,-179.9982,0.0043,0.0000
C00570=-90.851,41.782,4.400,-179.9836,0.0356,0.0000
C00571=-89.625,44.332,4.399,-179.8915,0.2161,0.0000
C00572=-88.233,46.990,4.399,-179.5895,0.7516,0.0000
C00573=-86.848,49.428,4.399,-179.0907,1.5395,0.0000
C00574=-85.672,51.352,4.398,-178.4158,2.4923,0.0000
C00575=-84.692,52.853,4.396,-177.6021,3.5812,0.0000
C00576=-83.700,54.314,4.393,-176.7898,4.6682,0.0000
C00577=-82.455,56.108,4.390,-176.0730,5.5771,0.0000
C00578=-80.608,58.679,4.388,-175.4847,6.1227,0.0000
C00579=-77.804,62.331,4.387,-175.0460,6.1652,0.0000
C00580=-74.450,66.299,4.387,-174.7278,5.9189,0.0000
C00581=-70.493,70.493,4.387,-174.3980,5.6020,0.0000
C00582=-66.299,74.450,4.387,-174.0812,5.2722,0.0000
C00583=-62.331,77.804,4.387,-173.8348,4.9540,0.0000
C00584=-58.679,80.608,4.388,-173.8773,4.5153,0.0000
C00585=-56.108,82.455,4.390,-174.4229,3.9270,0.0000
C00586=-54.314,83.700,4.393,-175.3318,3.2102,0.0000
C00587=-52.853,84.692,4.396,-176.4188,2.3979,0.0000
C00588=-51.352,85.672,4.398,-177.5077,1.5842,0.0000
C00589=-49.428,86.848,4.399,-178.4605,0.9093,0.0000
C00590=-46.990,88.233,4.399,-179.2484,0.4105,0.0000
C00591=-44.332,89.625,4.399,-179.7839,0.1085,0.0000
C00592=-41.782,90.851,4.400,-179.9644,0.0164,0.0000
C00593=-39.424,91.901,4.400,-179.9957,0.0018,0.0000
C00594=-37.107,92.860,4.400,-179.9957,0.0017,0.0000
C00595=-34.697,93.786,4.400,-179.9632,0.0136,0.0000
C00596=-32.027,94.722,4.399,-179.7705,0.0761,0.0000
C00597=-29.164,95.617,4.399,-179.1783,0.2412,0.0000
C00598=-26.460,96.362,4.399,-178.2686,0.4458,0.0000
C00599=-24.268,96.890,4.398,-177.1185,0.6429,0.0000
C00600=-22.514,97.259,4.396,-175.7755,0.8390,0.0000
C00601=-20.779,97.591,4.393,-174.4370,1.0358,0.0000
C00602=-18.630,97.979,4.390,-173.2935,1.1748,0.0000
C00603=-15.506,98.490,4.388,-172.4978,1.1464,0.0000
C00604=-10.941,99.090,4.387,-172.1612,0.8645,0.0000
C00605=-5.764,99.524,4.387,-172.1115,0.4617,0.0000
C00606=0.000,99.691,4.387,-172.1026,0.0000,0.0000
C00607=0.000,99.321,6.555,-168.5288,0.0000,0.0000
C00608=5.730,99.155,6.555,-168.5414,-0.6746,0.0000
C00609=10.884,98.723,6.555,-168.6119,-1.2518,0.0000
C00610=15.437,98.140,6.558,-169.0875,-1.6029,0.0000
C00611=18.547,97.668,6.566,-170.2252,-1.5293,0.0000
C00612=20.687,97.336,6.576,-171.8906,-1.2412,0.0000
C00613=22.417,97.071,6.585,-173.8606,-0.9699,0.0000
C00614=24.167,96.770,6.592,-175.8319,-0.7885,0.0000
C00615=26.351,96.303,6.595,-177.5102,-0.5868,0.0000
C00616=29.062,95.605,6.597,-178.8311,-0.3259,0.0000
C00617=31.947,94.737,6.598,-179.6815,-0.1030,0.0000
C00618=34.646,93.803,6.599,-179.9483,-0.0190,0.0000
C00619=37.090,92.867,6.600,-179.9940,-0.0024,0.0000
C00620=39.440,91.893,6.600,-179.9940,-0.0026,0.0000
C00621=41.830,90.827,6.599,-179.9500,-0.0231,0.0000
C00622=44.399,89.579,6.598,-179.7019,-0.1524,0.0000
C00623=47.053,88.152,6.597,-178.9430,-0.5962,0.0000
C00624=49.464,86.729,6.595,-177.8245,-1.3465,0.0000
C00625=51.338,85.515,6.592,-176.4942,-2.3935,0.0000
C00626=52.788,84.491,6.585,-174.9692,-3.6670,0.0000
C00627=54.199,83.455,6.576,-173.3790,-4.8831,0.0000
C00628=55.947,82.176,6.566,-171.9912,-5.8773,0.0000
C00629=58.480,80.311,6.558,-171.1269,-6.6473,0.0000
C00630=62.112,77.504,6.555,-171.0284,-7.2364,0.0000
C00631=66.061,74.165,6.555,-171.3764,-7.6887,0.0000
C00632=70.230,70.230,6.555,-171.8342,-8.1658,0.0000
C00633=74.165,66.061,6.555,-172.3113,-8.6235,0.0000
C00634=77.504,62.112,6.555,-172.7636,-8.9716,0.0000
C00635=80.311,58.480,6.558,-173.3528,-8.8731,0.0000
C00636=82.176,55.947,6.566,-174.1227,-8.0088,0.0000
C00637=83.455,54.199,6.576,-175.1169,-6.6210,0.0000
C00638=84.491,52.788,6.585,-176.3330,-5.0308,0.0000
C00639=85.515,51.338,6.592,-177.6065,-3.5058,0.0000
C00640=86.729,49.464,6.595,-178.6535,-2.1755,0.0000
C00641=88.152,47.053,6.597,-179.4038,-1.0570,0.0000
C00642=89.579,44.399,6.598,-179.8476,-0.2981,0.0000
C00643=90.827,41.830,6.599,-179.9769,-0.0500,0.0000
C00644=91.893,39.440,6.600,-179.9974,-0.0060,0.0000
C00645=92.867,37.090,6.600,-179.9976,-0.0060,0.0000
C00646=93.803,34.646,6.599,-179.9810,-0.0517,0.0000
C00647=94.737,31.947,6.598,-179.8970,-0.3185,0.0000
C00648=95.605,29.062,6.597,-179.6741,-1.1689,0.0000
C00649=96.303,26.351,6.595,-179.4132,-2.4898,0.0000
C00650=96.770,24.167,6.592,-179.2115,-4.1681,0.0000
C00651=97.071,22.417,6.585,-179.0301,-6.1394,0.0000
C00652=97.336,20.687,6.576,-178.7588,-8.1094,0.0000
C00653=97.668,18.547,6.566,-178.4707,-9.7748,0.0000
C00654=98.140,15.437,6.558,-178.3971,-10.9125,0.0000
C00655=98.723,10.884,6.555,-178.7482,-11.3881,0.0000
C00656=99.155,5.730,6.555,-179.3254,-11.4586,0.0000
C00657=99.321,0.000,6.555,180.0000,-11.4712,0.0000
C00658=99.155,-5.730,6.555,179.3254,-11.4585,0.0000
C00659=98.723,-10.884,6.555,178.7482,-11.3882,0.0000
C00660=98.140,-15.437,6.558,178.3971,-10.9125,0.0000
C00661=97.668,-18.547,6.566,178.4707,-9.7748,0.0000
C00662=97.336,-20.687,6.576,178.7588,-8.1094,0.0000
C00663=97.071,-22.417,6.585,179.0301,-6.1394,0.0000
C00664=96.770,-24.167,6.592,179.2115,-4.1681,0.0000
C00665=96.303,-26.351,6.595,179.4132,-2.4898,0.0000
C00666=95.605,-29.062,6.597,179.6741,-1.1689,0.0000
C00667=94.737,-31.947,6.598,179.8970,-0.3185,0.0000
C00668=93.803,-34.646,6.599,179.9810,-0.0517,0.0000
C00669=92.867,-37.090,6.600,179.9976,-0.0060,0.0000
C00670=91.893,-39.440,6.600,179.9974,-0.0060,0.0000
C00671=90.827,-41.830,6.599,179.9769,-0.0500,0.0000
C00672=89.579,-44.399,6.598,179.8476,-0.2981,0.0000
C00673=88.152,-47.053,6.597,179.4038,-1.0570,0.0000
C00674=86.729,-49.464,6.595,178.6535,-2.1755,0.0000
C00675=85.515,-51.338,6.592,177.6065,-3.5058,0.0000
C00676=84.491,-52.788,6.585,176.3330,-5.0308,0.0000
C00677=83.455,-54.199,6.576,175.1169,-6.6210,0.0000
C00678=82.176,-55.947,6.566,174.1227,-8.0088,0.0000
C00679=80.311,-58.480,6.558,173.3527,-8.8731,0.0000
C00680=77.504,-62.112,6.555,172.7636,-8.9716,0.0000
C00681=74.165,-66.061,6.555,172.3113,-8.6236,0.0000
C00682=70.230,-70.230,6.555,171.8342,-8.1658,0.0000
C00683=66.061,-74.165,6.555,171.3765,-7.6887,0.0000
C00684=62.112,-77.504,6.555,171.0284,-7.2364,0.0000
C00685=58.480,-80.311,6.558,171.1269,-6.6472,0.0000
C00686=55.947,-82.176,6.566,171.9912,-5.8773,0.0000
C00687=54.199,-83.455,6.576,173.3790,-4.8831,0.0000
C00688=52.788,-84.491,6.585,174.9692,-3.6670,0.0000
C00689=51.338,-85.515,6.592,176.4942,-2.3935,0.0000
C00690=49.464,-86.729,6.595,177.8245,-1.3465,0.0000
C00691=47.053,-88.152,6.597,178.9430,-0.5962,0.0000
C00692=44.399,-89.579,6.598,179.7019,-0.1524,0.0000
C00693=41.830,-90.827,6.599,179.9500,-0.0231,0.0000
C00694=39.440,-91.893,6.600,179.9940,-0.0026,0.0000
C00695=37.090,-92.867,6.600,179.9940,-0.0024,0.0000
C00696=34.646,-93.803,6.599,179.9483,-0.0190,0.0000
C00697=31.947,-94.737,6.598,179.6815,-0.1030,0.0000
C00698=29.062,-95.605,6.597,178.8311,-0.3259,0.0000
C00699=26.351,-96.303,6.595,177.5102,-0.5868,0.0000
C00700=24.167,-96.770,6.592,175.8319,-0.7885,0.0000
C00701=22.417,-97.071,6.585,173.8606,-0.9699,0.0000
C00702=20.687,-97.336,6.576,171.8906,-1.2412,0.0000
C00703=18.547,-97.668,6.566,170.2252,-1.5293,0.0000
C00704=15.437,-98.140,6.558,169.0875,-1.6029,0.0000
C00705=10.884,-98.723,6.555,168.6119,-1.2518,0.0000
C00706=5.730,-99.155,6.555,168.5414,-0.6746,0.0000
C00707=0.000,-99.321,6.555,168.5288,0.0000,0.0000
C00708=0.000,-99.321,6.555,168.5288,0.0000,0.0000
C00709=-5.730,-99.155,6.555,168.5415,0.6746,0.0000
C00710=-10.884,-98.723,6.555,168.6118,1.2518,0.0000
C00711=-15.437,-98.140,6.558,169.0875,1.6029,0.0000
C00712=-18.547,-97.668,6.566,170.2252,1.5293,0.0000
C00713=-20.687,-97.336,6.576,171.8906,1.2412,0.0000
C00714=-22.417,-97.071,6.585,173.8606,0.9699,0.0000
C00715=-24.167,-96.770,6.592,175.8319,0.7885,0.0000
C00716=-26.351,-96.303,6.595,177.5102,0.5868,0.0000
C00717=-29.062,-95.605,6.597,178.8311,0.3259,0.0000
C00718=-31.947,-94.737,6.598,179.6815,0.1030,0.0000
C00719=-34.646,-93.803,6.599,179.9483,0.0190,0.0000
C00720=-37.090,-92.867,6.600,179.9940,0.0024,0.0000
C00721=-39.440,-91.893,6.600,179.9940,0.0026,0.0000
C00722=-41.830,-90.827,6.599,179.9500,0.0231,0.0000
C00723=-44.399,-89.579,6.598,179.7019,0.1524,0.0000
C00724=-47.053,-88.152,6.597,178.9430,0.5962,0.0000
C00725=-49.464,-86.729,6.595,177.8245,1.3465,0.0000
C00726=-51.338,-85.515,6.592,176.4942,2.3935,0.0000
C00727=-52.788,-84.491,6.585,174.9692,3.6670,0.0000
C00728=-54.199,-83.455,6.576,173.3790,4.8831,0.0000
C00729=-55.947,-82.176,6.566,171.9912,5.8773,0.0000
C00730=-58.480,-80.311,6.558,171.1269,6.6473,0.0000
C00731=-62.112,-77.504,6.555,171.0284,7.2364,0.0000
C00732=-66.061,-74.165,6.555,171.3764,7.6887,0.0000
C00733=-70.230,-70.230,6.555,171.8342,8.1658,0.0000
C00734=-74.165,-66.061,6.555,172.3113,8.6235,0.0000
C00735=-77.504,-62.112,6.555,172.7636,8.9716,0.0000
C00736=-80.311,-58.480,6.558,173.3528,8.8731,0.0000
C00737=-82.176,-55.947,6.566,174.1227,8.0088,0.0000
C00738=-83.455,-54.199,6.576,175.1169,6.6210,0.0000
C00739=-84.491,-52.788,6.585,176.3330,5.0308,0.0000
C00740=-85.515,-51.338,6.592,177.6065,3.5058,0.0000
C00741=-86.729,-49.464,6.595,178.6535,2.1755,0.0000
C00742=-88.152,-47.053,6.597,179.4038,1.0570,0.0000
C00743=-89.579,-44.399,6.598,179.8476,0.2981,0.0000
C00744=-90.827,-41.830,6.599,179.9769,0.0500,0.0000
C00745=-91.893,-39.440,6.600,179.9974,0.0060,0.0000
C00746=-92.867,-37.090,6.600,179.9976,0.0060,0.0000
C00747=-93.803,-34.646,6.599,179.9810,0.0517,0.0000
C00748=-94.737,-31.947,6.598,179.8970,0.3185,0.0000
C00749=-95.605,-29.062,6.597,179.6741,1.1689,0.0000
C00750=-96.303,-26.351,6.595,179.4132,2.4898,0.0000
C00751=-96.770,-24.167,6.592,179.2115,4.1681,0.0000
C00752=-97.071,-22.417,6.585,179.0301,6.1394,0.0000
C00753=-97.336,-20.687,6.576,178.7588,8.1094,0.0000
C00754=-97.668,-18.547,6.566,178.4707,9.7748,0.0000
C00755=-98.140,-15.437,6.558,178.3971,10.9125,0.0000
C00756=-98.723,-10.884,6.555,178.7482,11.3881,0.0000
C00757=-99.155,-5.730,6.555,179.3254,11.4586,0.0000
C00758=-99.321,0.000,6.555,-180.0000,11.4712,0.0000
C00759=-99.155,5.730,6.555,-179.3254,11.4585,0.0000
C00760=-98.723,10.884,6.555,-178.7482,11.3882,0.0000
C00761=-98.140,15.437,6.558,-178.3971,10.9125,0.0000
C00762=-97.668,18.547,6.566,-178.4707,9.7748,0.0000
C00763=-97.336,20.687,6.576,-178.7588,8.1094,0.0000
C00764=-97.071,22.417,6.585,-179.0301,6.1394,0.0000
C00765=-96.770,24.167,6.592,-179.2115,4.1681,0.0000
C00766=-96.303,26.351,6.595,-179.4132,2.4898,0.0000
C00767=-95.605,29.062,6.597,-179.6741,1.1689,0.0000
C00768=-94.737,31.947,6.598,-179.8970,0.3185,0.0000
C00769=-93.803,34.646,6.599,-179.9810,0.0517,0.0000
C00770=-92.867,37.090,6.600,-179.9976,0.0060,0.0000
C00771=-91.893,39.440,6.600,-179.9974,0.0060,0.0000
C00772=-90.827,41.830,6.599,-179.9769,0.0500,0.0000
C00773=-89.579,44.399,6.598,-179.8476,0.2981,0.0000
C00774=-88.152,47.053,6.597,-179.4038,1.0570,0.0000
C00775=-86.729,49.464,6.595,-178.6535,2.1755,0.0000
C00776=-85.515,51.338,6.592,-177.6065,3.5058,0.0000
C00777=-84.491,52.788,6.585,-176.3330,5.0308,0.0000
C00778=-83.455,54.199,6.576,-175.1169,6.6210,0.0000
C00779=-82.176,55.947,6.566,-174.1227,8.0088,0.0000
C00780=-80.311,58.480,6.558,-173.3527,8.8731,0.0000
C00781=-77.504,62.112,6.555,-172.7636,8.9716,0.0000
C00782=-74.165,66.061,6.555,-172.3113,8.6236,0.0000
C00783=-70.230,70.230,6.555,-171.8342,8.1658,0.0000
C00784=-66.061,74.165,6.555,-171.3765,7.6887,0.0000
C00785=-62.112,77.504,6.555,-171.0284,7.2364,0.0000
C00786=-58.480,80.311,6.558,-171.1269,6.6472,0.0000
C00787=-55.947,82.176,6.566,-171.9912,5.8773,0.0000
C00788=-54.199,83.455,6.576,-173.3790,4.8831,0.0000
C00789=-52.788,84.491,6.585,-174.9692,3.6670,0.0000
C00790=-51.338,85.515,6.592,-176.4942,2.3935,0.0000
C00791=-49.464,86.729,6.595,-177.8245,1.3465,0.0000
C00792=-47.053,88.152,6.597,-178.9430,0.5962,0.0000
C00793=-44.399,89.579,6.598,-179.7019,0.1524,0.0000
C00794=-41.830,90.827,6.599,-179.9500,0.0231,0.0000
C00795=-39.440,91.893,6.600,-179.9940,0.0026,0.0000
C00796=-37.090,92.867,6.600,-179.9940,0.0024,0.0000
C00797=-34.646,93.803,6.599,-179.9483,0.0190,0.0000
C00798=-31.947,94.737,6.598,-179.6815,0.1030,0.0000
C00799=-29.062,95.605,6.597,-178.8311,0.3259,0.0000
C00800=-26.351,96.303,6.595,-177.5102,0.5868,0.0000
C00801=-24.167,96.770,6.592,-175.8319,0.7885,0.0000
C00802=-22.417,97.071,6.585,-173.8606,0.9699,0.0000
C00803=-20.687,97.336,6.576,-171.8906,1.2412,0.0000
C00804=-18.547,97.668,6.566,-170.2252,1.5293,0.0000
C00805=-15.437,98.140,6.558,-169.0875,1.6029,0.0000
C00806=-10.884,98.723,6.555,-168.6118,1.2518,0.0000
C00807=-5.730,99.155,6.555,-168.5415,0.6746,0.0000
C00808=0.000,99.321,6.555,-168.5288,0.0000,0.0000
C00809=0.000,98.820,8.697,-165.2395,0.0000,0.0000
C00810=5.684,98.656,8.697,-165.2556,-0.8746,0.0000
C00811=10.807,98.229,8.698,-165.3433,-1.6024,0.0000
C00812=15.344,97.668,8.705,-165.9346,-1.9496,0.0000
C00813=18.436,97.247,8.723,-167.3796,-1.6454,0.0000
C00814=20.563,96.991,8.745,-169.5531,-1.1205,0.0000
C00815=22.286,96.814,8.767,-172.1394,-0.8021,0.0000
C00816=24.029,96.606,8.782,-174.6912,-0.7561,0.0000
C00817=26.202,96.222,8.789,-176.8486,-0.6486,0.0000
C00818=28.922,95.588,8.792,-178.5415,-0.3776,0.0000
C00819=31.837,94.757,8.795,-179.6165,-0.1196,0.0000
C00820=34.577,93.826,8.798,-179.9364,-0.0233,0.0000
C00821=37.066,92.876,8.800,-179.9926,-0.0029,0.0000
C00822=39.463,91.883,8.800,-179.9927,-0.0031,0.0000
C00823=41.895,90.794,8.798,-179.9386,-0.0286,0.0000
C00824=44.491,89.515,8.795,-179.6442,-0.1866,0.0000
C00825=47.140,88.042,8.792,-178.7017,-0.7645,0.0000
C00826=49.511,86.567,8.789,-177.3127,-1.7714,0.0000
C00827=51.320,85.302,8.782,-175.7087,-3.2266,0.0000
C00828=52.699,84.217,8.767,-173.8629,-5.0134,0.0000
C00829=54.043,83.124,8.745,-171.7941,-6.6477,0.0000
C00830=55.728,81.800,8.723,-169.8719,-7.8577,0.0000
C00831=58.212,79.911,8.705,-168.6223,-8.7038,0.0000
C00832=61.817,77.101,8.698,-168.4305,-9.3780,0.0000
C00833=65.741,73.780,8.697,-168.8617,-9.9428,0.0000
C00834=69.877,69.877,8.697,-169.4466,-10.5535,0.0000
C00835=73.780,65.741,8.697,-170.0572,-11.1383,0.0000
C00836=77.101,61.817,8.698,-170.6220,-11.5695,0.0000
C00837=79.911,58.212,8.705,-171.2962,-11.3776,0.0000
C00838=81.800,55.728,8.723,-172.1423,-10.1281,0.0000
C00839=83.124,54.043,8.745,-173.3523,-8.2059,0.0000
C00840=84.217,52.699,8.767,-174.9866,-6.1371,0.0000
C00841=85.302,51.320,8.782,-176.7734,-4.2913,0.0000
C00842=86.567,49.511,8.789,-178.2286,-2.6873,0.0000
C00843=88.042,47.140,8.792,-179.2355,-1.2983,0.0000
C00844=89.515,44.491,8.795,-179.8134,-0.3558,0.0000
C00845=90.794,41.895,8.798,-179.9714,-0.0614,0.0000
C00846=91.883,39.463,8.800,-179.9969,-0.0073,0.0000
C00847=92.876,37.066,8.800,-179.9971,-0.0074,0.0000
C00848=93.826,34.577,8.798,-179.9767,-0.0636,0.0000
C00849=94.757,31.837,8.795,-179.8804,-0.3835,0.0000
C00850=95.588,28.922,8.792,-179.6224,-1.4585,0.0000
C00851=96.222,26.202,8.789,-179.3514,-3.1514,0.0000
C00852=96.606,24.029,8.782,-179.2439,-5.3088,0.0000
C00853=96.814,22.286,8.767,-179.1979,-7.8606,0.0000
C00854=96.991,20.563,8.745,-178.8795,-10.4469,0.0000
C00855=97.247,18.436,8.723,-178.3546,-12.6204,0.0000
C00856=97.668,15.344,8.705,-178.0504,-14.0654,0.0000
C00857=98.229,10.807,8.698,-178.3976,-14.6567,0.0000
C00858=98.656,5.684,8.697,-179.1254,-14.7444,0.0000
C00859=98.820,0.000,8.697,180.0000,-14.7605,0.0000
C00860=98.656,-5.684,8.697,179.1254,-14.7444,0.0000
C00861=98.229,-10.807,8.698,178.3976,-14.6567,0.0000
C00862=97.668,-15.344,8.705,178.0504,-14.0654,0.0000
C00863=97.247,-18.436,8.723,178.3546,-12.6204,0.0000
C00864=96.991,-20.563,8.745,178.8795,-10.4469,0.0000
C00865=96.814,-22.286,8.767,179.1979,-7.8606,0.0000
C00866=96.606,-24.029,8.782,179.2439,-5.3088,0.0000
C00867=96.222,-26.202,8.789,179.3514,-3.1514,0.0000
C00868=95.588,-28.922,8.792,179.6224,-1.4585,0.0000
C00869=94.757,-31.837,8.795,179.8804,-0.3835,0.0000
C00870=93.826,-34.577,8.798,179.9767,-0.0636,0.0000
C00871=92.876,-37.066,8.800,179.9971,-0.0074,0.0000
C00872=91.883,-39.463,8.800,179.9969,-0.0073,0.0000
C00873=90.794,-41.895,8.798,179.9714,-0.0614,0.0000
C00874=89.515,-44.491,8.795,179.8134,-0.3558,0.0000
C00875=88.042,-47.140,8.792,179.2355,-1.2983,0.0000
C00876=86.567,-49.511,8.789,178.2286,-2.6873,0.0000
C00877=85.302,-51.320,8.782,176.7734,-4.2913,0.0000
C00878=84.217,-52.699,8.767,174.9866,-6.1371,0.0000
C00879=83.124,-54.043,8.745,173.3523,-8.2059,0.0000
C00880=81.800,-55.728,8.723,172.1423,-10.1281,0.0000
C00881=79.911,-58.212,8.705,171.2962,-11.3777,0.0000
C00882=77.101,-61.817,8.698,170.6220,-11.5695,0.0000
C00883=73.780,-65.741,8.697,170.0572,-11.1383,0.0000
C00884=69.877,-69.877,8.697,169.4465,-10.5534,0.0000
C00885=65.741,-73.780,8.697,168.8617,-9.9428,0.0000
C00886=61.817,-77.101,8.698,168.4305,-9.3780,0.0000
C00887=58.212,-79.911,8.705,168.6224,-8.7038,0.0000
C00888=55.728,-81.800,8.723,169.8719,-7.8577,0.0000
C00889=54.043,-83.124,8.745,171.7941,-6.6477,0.0000
C00890=52.699,-84.217,8.767,173.8629,-5.0134,0.0000
C00891=51.320,-85.302,8.782,175.7087,-3.2266,0.0000
C00892=49.511,-86.567,8.789,177.3127,-1.7714,0.0000
C00893=47.140,-88.042,8.792,178.7017,-0.7645,0.0000
C00894=44.491,-89.515,8.795,179.6442,-0.1866,0.0000
C00895=41.895,-90.794,8.798,179.9386,-0.0286,0.0000
C00896=39.463,-91.883,8.800,179.9927,-0.0031,0.0000
C00897=37.066,-92.876,8.800,179.9926,-0.0029,0.0000
C00898=34.577,-93.826,8.798,179.9364,-0.0233,0.0000
C00899=31.837,-94.757,8.795,179.6165,-0.1196,0.0000
C00900=28.922,-95.588,8.792,178.5415,-0.3776,0.0000
C00901=26.202,-96.222,8.789,176.8486,-0.6486,0.0000
C00902=24.029,-96.606,8.782,174.6912,-0.7561,0.0000
C00903=22.286,-96.814,8.767,172.1394,-0.8021,0.0000
C00904=20.563,-96.991,8.745,169.5531,-1.1205,0.0000
C00905=18.436,-97.247,8.723,167.3796,-1.6454,0.0000
C00906=15.344,-97.668,8.705,165.9346,-1.9496,0.0000
C00907=10.807,-98.229,8.698,165.3433,-1.6024,0.0000
C00908=5.684,-98.656,8.697,165.2556,-0.8746,0.0000
C00909=0.000,-98.820,8.697,165.2395,0.0000,0.0000
C00910=0.000,-98.820,8.697,165.2395,0.0000,0.0000
C00911=-5.684,-98.656,8.697,165.2556,0.8746,0.0000
C00912=-10.807,-98.229,8.698,165.3433,1.6024,0.0000
C00913=-15.344,-97.668,8.705,165.9346,1.9496,0.0000
C00914=-18.436,-97.247,8.723,167.3796,1.6454,0.0000
C00915=-20.563,-96.991,8.745,169.5531,1.1205,0.0000
C00916=-22.286,-96.814,8.767,172.1394,0.8021,0.0000
C00917=-24.029,-96.606,8.782,174.6912,0.7561,0.0000
C00918=-26.202,-96.222,8.789,176.8486,0.6486,0.0000
C00919=-28.922,-95.588,8.792,178.5415,0.3776,0.0000
C00920=-31.837,-94.757,8.795,179.6165,0.1196,0.0000
C00921=-34.577,-93.826,8.798,179.9364,0.0233,0.0000
C00922=-37.066,-92.876,8.800,179.9926,0.0029,0.0000
C00923=-39.463,-91.883,8.800,179.9927,0.0031,0.0000
C00924=-41.895,-90.794,8.798,179.9386,0.0286,0.0000
C00925=-44.491,-89.515,8.795,179.6442,0.1866,0.0000
C00926=-47.140,-88.042,8.792,178.7017,0.7645,0.0000
C00927=-49.511,-86.567,8.789,177.3127,1.7714,0.0000
C00928=-51.320,-85.302,8.782,175.7087,3.2266,0.0000
C00929=-52.699,-84.217,8.767,173.8629,5.0134,0.0000
C00930=-54.043,-83.124,8.745,171.7941,6.6477,0.0000
C00931=-55.728,-81.800,8.723,169.8719,7.8577,0.0000
C00932=-58.212,-79.911,8.705,168.6223,8.7038,0.0000
C00933=-61.817,-77.101,8.698,168.4305,9.3780,0.0000
C00934=-65.741,-73.780,8.697,168.8617,9.9428,0.0000
C00935=-69.877,-69.877,8.697,169.4466,10.5535,0.0000
C00936=-73.780,-65.741,8.697,170.0572,11.1383,0.0000
C00937=-77.101,-61.817,8.698,170.6220,11.5695,0.0000
C00938=-79.911,-58.212,8.705,171.2962,11.3776,0.0000
C00939=-81.800,-55.728,8.723,172.1423,10.1281,0.0000
C00940=-83.124,-54.043,8.745,173.3523,8.2059,0.0000
C00941=-84.217,-52.699,8.767,174.9866,6.1371,0.0000
C00942=-85.302,-51.320,8.782,176.7734,4.2913,0.0000
C00943=-86.567,-49.511,8.789,178.2286,2.6873,0.0000
C00944=-88.042,-47.140,8.792,179.2355,1.2983,0.0000
C00945=-89.515,-44.491,8.795,179.8134,0.3558,0.0000
C00946=-90.794,-41.895,8.798,179.9714,0.0614,0.0000
C00947=-91.883,-39.463,8.800,179.9969,0.0073,0.0000
C00948=-92.876,-37.066,8.800,179.9971,0.0074,0.0000
C00949=-93.826,-34.577,8.798,179.9767,0.0636,0.0000
C00950=-94.757,-31.837,8.795,179.8804,0.3835,0.0000
C00951=-95.588,-28.922,8.792,179.6224,1.4585,0.0000
C00952=-96.222,-26.202,8.789,179.3514,3.1514,0.0000
C00953=-96.606,-24.029,8.782,179.2439,5.3088,0.0000
C00954=-96.814,-22.286,8.767,179.1979,7.8606,0.0000
C00955=-96.991,-20.563,8.745,178.8795,10.4469,0.0000
C00956=-97.247,-18.436,8.723,178.3546,12.6204,0.0000
C00957=-97.668,-15.344,8.705,178.0504,14.0654,0.0000
C00958=-98.229,-10.807,8.698,178.3976,14.6567,0.0000
C00959=-98.656,-5.684,8.697,179.1254,14.7444,0.0000
C00960=-98.820,0.000,8.697,-180.0000,14.7605,0.0000
C00961=-98.656,5.684,8.697,-179.1254,14.7444,0.0000
C00962=-98.229,10.807,8.698,-178.3976,14.6567,0.0000
C00963=-97.668,15.344,8.705,-178.0504,14.0654,0.0000
C00964=-97.247,18.436,8.723,-178.3546,12.6204,0.0000
C00965=-96.991,20.563,8.745,-178.8795,10.4469,0.0000
C00966=-96.814,22.286,8.767,-179.1979,7.8606,0.0000
C00967=-96.606,24.029,8.782,-179.2439,5.3088,0.0000
C00968=-96.222,26.202,8.789,-179.3514,3.1514,0.0000
C00969=-95.588,28.922,8.792,-179.6224,1.4585,0.0000
C00970=-94.757,31.837,8.795,-179.8804,0.3835,0.0000
C00971=-93.826,34.577,8.798,-179.9767,0.0636,0.0000
C00972=-92.876,37.066,8.800,-179.9971,0.0074,0.0000
C00973=-91.883,39.463,8.800,-179.9969,0.0073,0.0000
C00974=-90.794,41.895,8.798,-179.9714,0.0614,0.0000
C00975=-89.515,44.491,8.795,-179.8134,0.3558,0.0000
C00976=-88.042,47.140,8.792,-179.2355,1.2983,0.0000
C00977=-86.567,49.511,8.789,-178.2286,2.6873,0.0000
C00978=-85.302,51.320,8.782,-176.7734,4.2913,0.0000
C00979=-84.217,52.699,8.767,-174.9866,6.1371,0.0000
C00980=-83.124,54.043,8.745,-173.3523,8.2059,0.0000
C00981=-81.800,55.728,8.723,-172.1423,10.1281,0.0000
C00982=-79.911,58.212,8.705,-171.2962,11.3777,0.0000
C00983=-77.101,61.817,8.698,-170.6220,11.5695,0.0000
C00984=-73.780,65.741,8.697,-170.0572,11.1383,0.0000
C00985=-69.877,69.877,8.697,-169.4465,10.5534,0.0000
C00986=-65.741,73.780,8.697,-168.8617,9.9428,0.0000
C00987=-61.817,77.101,8.698,-168.4305,9.3780,0.0000
C00988=-58.212,79.911,8.705,-168.6224,8.7038,0.0000
C00989=-55.728,81.800,8.723,-169.8719,7.8577,0.0000
C00990=-54.043,83.124,8.745,-171.7941,6.6477,0.0000
C00991=-52.699,84.217,8.767,-173.8629,5.0134,0.0000
C00992=-51.320,85.302,8.782,-175.7087,3.2266,0.0000
C00993=-49.511,86.567,8.789,-177.3127,1.7714,0.0000
C00994=-47.140,88.042,8.792,-178.7017,0.7645,0.0000
C00995=-44.491,89.515,8.795,-179.6442,0.1866,0.0000
C00996=-41.895,90.794,8.798,-179.9386,0.0286,0.0000
C00997=-39.463,91.883,8.800,-179.9927,0.0031,0.0000
C00998=-37.066,92.876,8.800,-179.9926,0.0029,0.0000
C00999=-34.577,93.826,8.798,-179.9364,0.0233,0.0000
C01000=-31.837,94.757,8.795,-179.6165,0.1196,0.0000
C01001=-28.922,95.588,8.792,-178.5415,0.3776,0.0000
C01002=-26.202,96.222,8.789,-176.8486,0.6486,0.0000
C01003=-24.029,96.606,8.782,-174.6912,0.7561,0.0000
C01004=-22.286,96.814,8.767,-172.1394,0.8021,0.0000
C01005=-20.563,96.991,8.745,-169.5531,1.1205,0.0000
C01006=-18.436,97.247,8.723,-167.3796,1.6454,0.0000
C01007=-15.344,97.668,8.705,-165.9346,1.9496,0.0000
C01008=-10.807,98.229,8.698,-165.3433,1.6024,0.0000
C01009=-5.684,98.656,8.697,-165.2556,0.8746,0.0000
C01010=0.000,98.820,8.697,-165.2395,0.0000,0.0000
C01011=0.000,98.204,10.809,-162.2405,0.0001,0.0000
C01012=5.628,98.041,10.809,-162.2594,-1.0613,0.0000
C01013=10.712,97.620,10.809,-162.3610,-1.9132,0.0000
C01014=15.229,97.084,10.823,-163.0467,-2.1695,0.0000
C01015=18.298,96.727,10.856,-164.7843,-1.4750,0.0000
C01016=20.409,96.562,10.898,-167.4920,-0.6133,0.0000
C01017=22.123,96.495,10.937,-170.6949,-0.2914,0.0000
C01018=23.856,96.400,10.965,-173.7465,-0.5203,0.0000
C01019=26.016,96.121,10.978,-176.3051,-0.6217,0.0000
C01020=28.748,95.567,10.985,-178.3192,-0.3939,0.0000
C01021=31.699,94.782,10.991,-179.5791,-0.1255,0.0000
C01022=34.490,93.854,10.996,-179.9278,-0.0262,0.0000
C01023=37.037,92.887,11.000,-179.9917,-0.0033,0.0000
C01024=39.492,91.870,11.000,-179.9918,-0.0035,0.0000
C01025=41.977,90.753,10.996,-179.9305,-0.0325,0.0000
C01026=44.606,89.436,10.991,-179.6137,-0.2089,0.0000
C01027=47.248,87.904,10.985,-178.5329,-0.9103,0.0000
C01028=49.571,86.364,10.978,-176.9470,-2.1756,0.0000
C01029=51.296,85.034,10.965,-175.2038,-4.0647,0.0000
C01030=52.589,83.875,10.937,-173.1881,-6.4053,0.0000
C01031=53.849,82.711,10.898,-170.6621,-8.4913,0.0000
C01032=55.458,81.334,10.856,-168.1110,-9.8772,0.0000
C01033=57.880,79.417,10.823,-166.3774,-10.6897,0.0000
C01034=61.453,76.603,10.809,-166.0469,-11.3770,0.0000
C01035=65.346,73.305,10.809,-166.5413,-12.0309,0.0000
C01036=69.440,69.440,10.809,-167.2392,-12.7609,0.0000
C01037=73.305,65.346,10.809,-167.9691,-13.4586,0.0000
C01038=76.603,61.453,10.809,-168.6230,-13.9530,0.0000
C01039=79.417,57.880,10.823,-169.3103,-13.6226,0.0000
C01040=81.334,55.458,10.856,-170.1228,-11.8890,0.0000
C01041=82.711,53.849,10.898,-171.5087,-9.3379,0.0000
C01042=83.875,52.589,10.937,-173.5947,-6.8119,0.0000
C01043=85.034,51.296,10.965,-175.9353,-4.7962,0.0000
C01044=86.364,49.571,10.978,-177.8244,-3.0530,0.0000
C01045=87.904,47.248,10.985,-179.0897,-1.4671,0.0000
C01046=89.436,44.606,10.991,-179.7911,-0.3863,0.0000
C01047=90.753,41.977,10.996,-179.9675,-0.0695,0.0000
C01048=91.870,39.492,11.000,-179.9965,-0.0082,0.0000
C01049=92.887,37.037,11.000,-179.9967,-0.0083,0.0000
C01050=93.854,34.490,10.996,-179.9738,-0.0722,0.0000
C01051=94.782,31.699,10.991,-179.8745,-0.4209,0.0000
C01052=95.567,28.748,10.985,-179.6061,-1.6808,0.0000
C01053=96.121,26.016,10.978,-179.3783,-3.6949,0.0000
C01054=96.400,23.856,10.965,-179.4797,-6.2535,0.0000
C01055=96.495,22.123,10.937,-179.7086,-9.3051,0.0000
C01056=96.562,20.409,10.898,-179.3867,-12.5080,0.0000
C01057=96.727,18.298,10.856,-178.5250,-15.2157,0.0000
C01058=97.084,15.229,10.823,-177.8305,-16.9533,0.0000
C01059=97.620,10.712,10.809,-178.0868,-17.6390,0.0000
C01060=98.041,5.628,10.809,-178.9387,-17.7406,0.0000
C01061=98.204,0.000,10.809,179.9999,-17.7595,0.0000
C01062=98.041,-5.628,10.809,178.9388,-17.7405,0.0000
C01063=97.620,-10.712,10.809,178.0869,-17.6390,0.0000
C01064=97.084,-15.229,10.823,177.8304,-16.9533,0.0000
C01065=96.727,-18.298,10.856,178.5250,-15.2157,0.0000
C01066=96.562,-20.409,10.898,179.3867,-12.5080,0.0000
C01067=96.495,-22.123,10.937,179.7086,-9.3051,0.0000
C01068=96.400,-23.856,10.965,179.4797,-6.2535,0.0000
C01069=96.121,-26.016,10.978,179.3783,-3.6949,0.0000
C01070=95.567,-28.748,10.985,179.6061,-1.6808,0.0000
C01071=94.782,-31.699,10.991,179.8745,-0.4209,0.0000
C01072=93.854,-34.490,10.996,179.9738,-0.0722,0.0000
C01073=92.887,-37.037,11.000,179.9967,-0.0083,0.0000
C01074=91.870,-39.492,11.000,179.9965,-0.0082,0.0000
C01075=90.753,-41.977,10.996,179.9675,-0.0695,0.0000
C01076=89.436,-44.606,10.991,179.7911,-0.3863,0.0000
C01077=87.904,-47.248,10.985,179.0897,-1.4671,0.0000
C01078=86.364,-49.571,10.978,177.8244,-3.0530,0.0000
C01079=85.034,-51.296,10.965,175.9353,-4.7962,0.0000
C01080=83.875,-52.589,10.937,173.5947,-6.8119,0.0000
C01081=82.711,-53.849,10.898,171.5087,-9.3379,0.0000
C01082=81.334,-55.458,10.856,170.1228,-11.8890,0.0000
C01083=79.417,-57.880,10.823,169.3103,-13.6226,0.0000
C01084=76.603,-61.453,10.809,168.6230,-13.9531,0.0000
C01085=73.305,-65.346,10.809,167.9691,-13.4587,0.0000
C01086=69.440,-69.440,10.809,167.2391,-12.7608,0.0000
C01087=65.346,-73.305,10.809,166.5414,-12.0309,0.0000
C01088=61.453,-76.603,10.809,166.0470,-11.3770,0.0000
C01089=57.880,-79.417,10.823,166.3774,-10.6897,0.0000
C01090=55.458,-81.334,10.856,168.1110,-9.8772,0.0000
C01091=53.849,-82.711,10.898,170.6621,-8.4913,0.0000
C01092=52.589,-83.875,10.937,173.1881,-6.4053,0.0000
C01093=51.296,-85.034,10.965,175.2038,-4.0647,0.0000
C01094=49.571,-86.364,10.978,176.9470,-2.1756,0.0000
C01095=47.248,-87.904,10.985,178.5329,-0.9103,0.0000
C01096=44.606,-89.436,10.991,179.6137,-0.2089,0.0000
C01097=41.977,-90.753,10.996,179.9305,-0.0325,0.0000
C01098=39.492,-91.870,11.000,179.9918,-0.0035,0.0000
C01099=37.037,-92.887,11.000,179.9917,-0.0033,0.0000
C01100=34.490,-93.854,10.996,179.9278,-0.0262,0.0000
C01101=31.699,-94.782,10.991,179.5791,-0.1255,0.0000
C01102=28.748,-95.567,10.985,178.3192,-0.3939,0.0000
C01103=26.016,-96.121,10.978,176.3051,-0.6217,0.0000
C01104=23.856,-96.400,10.965,173.7465,-0.5203,0.0000
C01105=22.123,-96.495,10.937,170.6949,-0.2914,0.0000
C01106=20.409,-96.562,10.898,167.4920,-0.6133,0.0000
C01107=18.298,-96.727,10.856,164.7843,-1.4750,0.0000
C01108=15.229,-97.084,10.823,163.0467,-2.1695,0.0000
C01109=10.712,-97.620,10.809,162.3610,-1.9132,0.0000
C01110=5.628,-98.041,10.809,162.2594,-1.0613,0.0000
C01111=0.000,-98.204,10.809,162.2405,0.0001,0.0000
C01112=0.000,-98.204,10.809,162.2405,0.0001,0.0000
C01113=-5.628,-98.041,10.809,162.2595,1.0612,0.0000
C01114=-10.712,-97.620,10.809,162.3610,1.9131,0.0000
C01115=-15.229,-97.084,10.823,163.0467,2.1696,0.0000
C01116=-18.298,-96.727,10.856,164.7843,1.4750,0.0000
C01117=-20.409,-96.562,10.898,167.4920,0.6133,0.0000
C01118=-22.123,-96.495,10.937,170.6949,0.2914,0.0000
C01119=-23.856,-96.400,10.965,173.7465,0.5203,0.0000
C01120=-26.016,-96.121,10.978,176.3051,0.6217,0.0000
C01121=-28.748,-95.567,10.985,178.3192,0.3939,0.0000
C01122=-31.699,-94.782,10.991,179.5791,0.1255,0.0000
C01123=-34.490,-93.854,10.996,179.9278,0.0262,0.0000
C01124=-37.037,-92.887,11.000,179.9917,0.0033,0.0000
C01125=-39.492,-91.870,11.000,179.9918,0.0035,0.0000
C01126=-41.977,-90.753,10.996,179.9305,0.0325,0.0000
C01127=-44.606,-89.436,10.991,179.6137,0.2089,0.0000
C01128=-47.248,-87.904,10.985,178.5329,0.9103,0.0000
C01129=-49.571,-86.364,10.978,176.9470,2.1756,0.0000
C01130=-51.296,-85.034,10.965,175.2038,4.0647,0.0000
C01131=-52.589,-83.875,10.937,173.1881,6.4053,0.0000
C01132=-53.849,-82.711,10.898,170.6621,8.4913,0.0000
C01133=-55.458,-81.334,10.856,168.1110,9.8772,0.0000
C01134=-57.880,-79.417,10.823,166.3774,10.6897,0.0000
C01135=-61.453,-76.603,10.809,166.0469,11.3770,0.0000
C01136=-65.346,-73.305,10.809,166.5413,12.0309,0.0000
C01137=-69.440,-69.440,10.809,167.2392,12.7609,0.0000
C01138=-73.305,-65.346,10.809,167.9691,13.4586,0.0000
C01139=-76.603,-61.453,10.809,168.6230,13.9530,0.0000
C01140=-79.417,-57.880,10.823,169.3103,13.6226,0.0000
C01141=-81.334,-55.458,10.856,170.1228,11.8890,0.0000
C01142=-82.711,-53.849,10.898,171.5087,9.3379,0.0000
C01143=-83.875,-52.589,10.937,173.5947,6.8119,0.0000
C01144=-85.034,-51.296,10.965,175.9353,4.7962,0.0000
C01145=-86.364,-49.571,10.978,177.8244,3.0530,0.0000
C01146=-87.904,-47.248,10.985,179.0897,1.4671,0.0000
C01147=-89.436,-44.606,10.991,179.7911,0.3863,0.0000
C01148=-90.753,-41.977,10.996,179.9675,0.0695,0.0000
C01149=-91.870,-39.492,11.000,179.9965,0.0082,0.0000
C01150=-92.887,-37.037,11.000,179.9967,0.0083,0.0000
C01151=-93.854,-34.490,10.996,179.9738,0.0722,0.0000
C01152=-94.782,-31.699,10.991,179.8745,0.4209,0.0000
C01153=-95.567,-28.748,10.985,179.6061,1.6808,0.0000
C01154=-96.121,-26.016,10.978,179.3783,3.6949,0.0000
C01155=-96.400,-23.856,10.965,179.4797,6.2535,0.0000
C01156=-96.495,-22.123,10.937,179.7086,9.3051,0.0000
C01157=-96.562,-20.409,10.898,179.3867,12.5080,0.0000
C01158=-96.727,-18.298,10.856,178.5250,15.2157,0.0000
C01159=-97.084,-15.229,10.823,177.8305,16.9533,0.0000
C01160=-97.620,-10.712,10.809,178.0868,17.6390,0.0000
C01161=-98.041,-5.628,10.809,178.9387,17.7406,0.0000
C01162=-98.204,0.000,10.809,-179.9999,17.7595,0.0000
C01163=-98.041,5.628,10.809,-178.9388,17.7405,0.0000
C01164=-97.620,10.712,10.809,-178.0869,17.6390,0.0000
C01165=-97.084,15.229,10.823,-177.8304,16.9533,0.0000
C01166=-96.727,18.298,10.856,-178.5250,15.2157,0.0000
C01167=-96.562,20.409,10.898,-179.3867,12.5080,0.0000
C01168=-96.495,22.123,10.937,-179.7086,9.3051,0.0000
C01169=-96.400,23.856,10.965,-179.4797,6.2535,0.0000
C01170=-96.121,26.016,10.978,-179.3783,3.6949,0.0000
C01171=-95.567,28.748,10.985,-179.6061,1.6808,0.0000
C01172=-94.782,31.699,10.991,-179.8745,0.4209,0.0000
C01173=-93.854,34.490,10.996,-179.9738,0.0722,0.0000
C01174=-92.887,37.037,11.000,-179.9967,0.0083,0.0000
C01175=-91.870,39.492,11.000,-179.9965,0.0082,0.0000
C01176=-90.753,41.977,10.996,-179.9675,0.0695,0.0000
C01177=-89.436,44.606,10.991,-179.7911,0.3863,0.0000
C01178=-87.904,47.248,10.985,-179.0897,1.4671,0.0000
C01179=-86.364,49.571,10.978,-177.8244,3.0530,0.0000
C01180=-85.034,51.296,10.965,-175.9353,4.7962,0.0000
C01181=-83.875,52.589,10.937,-173.5947,6.8119,0.0000
C01182=-82.711,53.849,10.898,-171.5087,9.3379,0.0000
C01183=-81.334,55.458,10.856,-170.1228,11.8890,0.0000
C01184=-79.417,57.880,10.823,-169.3103,13.6226,0.0000
C01185=-76.603,61.453,10.809,-168.6230,13.9531,0.0000
C01186=-73.305,65.346,10.809,-167.9691,13.4587,0.0000
C01187=-69.440,69.440,10.809,-167.2391,12.7608,0.0000
C01188=-65.346,73.305,10.809,-166.5414,12.0309,0.0000
C01189=-61.453,76.603,10.809,-166.0470,11.3770,0.0000
C01190=-57.880,79.417,10.823,-166.3774,10.6897,0.0000
C01191=-55.458,81.334,10.856,-168.1110,9.8772,0.0000
C01192=-53.849,82.711,10.898,-170.6621,8.4913,0.0000
C01193=-52.589,83.875,10.937,-173.1881,6.4053,0.0000
C01194=-51.296,85.034,10.965,-175.2038,4.0647,0.0000
C01195=-49.571,86.364,10.978,-176.9470,2.1756,0.0000
C01196=-47.248,87.904,10.985,-178.5329,0.9103,0.0000
C01197=-44.606,89.436,10.991,-179.6137,0.2089,0.0000
C01198=-41.977,90.753,10.996,-179.9305,0.0325,0.0000
C01199=-39.492,91.870,11.000,-179.9918,0.0035,0.0000
C01200=-37.037,92.887,11.000,-179.9917,0.0033,0.0000
C01201=-34.490,93.854,10.996,-179.9278,0.0262,0.0000
C01202=-31.699,94.782,10.991,-179.5791,0.1255,0.0000
C01203=-28.748,95.567,10.985,-178.3192,0.3939,0.0000
C01204=-26.016,96.121,10.978,-176.3051,0.6217,0.0000
C01205=-23.856,96.400,10.965,-173.7465,0.5203,0.0000
C01206=-22.123,96.495,10.937,-170.6949,0.2914,0.0000
C01207=-20.409,96.562,10.898,-167.4920,0.6133,0.0000
C01208=-18.298,96.727,10.856,-164.7843,1.4750,0.0000
C01209=-15.229,97.084,10.823,-163.0467,2.1696,0.0000
C01210=-10.712,97.620,10.809,-162.3610,1.9131,0.0000
C01211=-5.628,98.041,10.809,-162.2595,1.0612,0.0000
C01212=0.000,98.204,10.809,-162.2405,0.0001,0.0000
C01213=0.000,97.482,12.888,-159.5253,0.0001,0.0000
C01214=5.562,97.322,12.887,-159.5467,-1.2345,0.0000
C01215=10.602,96.908,12.888,-159.6590,-2.1823,0.0000
C01216=15.094,96.401,12.910,-160.4230,-2.2510,0.0000
C01217=18.135,96.115,12.963,-162.4714,-0.9834,0.0000
C01218=20.227,96.057,13.031,-165.7975,0.3024,0.0000
C01219=21.929,96.117,13.096,-169.6348,0.5559,0.0000
C01220=23.652,96.157,13.142,-173.0616,-0.0823,0.0000
C01221=25.795,96.000,13.164,-175.9036,-0.5053,0.0000
C01222=28.540,95.542,13.175,-178.1724,-0.3760,0.0000
C01223=31.535,94.812,13.184,-179.5717,-0.1209,0.0000
C01224=34.387,93.888,13.193,-179.9229,-0.0278,0.0000
C01225=37.002,92.901,13.199,-179.9912,-0.0035,0.0000
C01226=39.526,91.855,13.199,-179.9913,-0.0038,0.0000
C01227=42.074,90.704,13.193,-179.9258,-0.0349,0.0000
C01228=44.743,89.341,13.184,-179.6117,-0.2174,0.0000
C01229=47.377,87.740,13.175,-178.4418,-1.0268,0.0000
C01230=49.643,86.123,13.164,-176.7447,-2.5426,0.0000
C01231=51.269,84.717,13.142,-175.0240,-4.8604,0.0000
C01232=52.459,83.471,13.096,-173.0176,-7.7557,0.0000
C01233=53.620,82.225,13.031,-170.0612,-10.3532,0.0000
C01234=55.140,80.787,12.963,-166.7496,-11.9257,0.0000
C01235=57.492,78.839,12.910,-164.3969,-12.6081,0.0000
C01236=61.028,76.021,12.888,-163.8761,-13.2352,0.0000
C01237=64.884,72.750,12.887,-164.4132,-13.9544,0.0000
C01238=68.930,68.930,12.888,-165.2103,-14.7899,0.0000
C01239=72.750,64.884,12.887,-166.0456,-15.5867,0.0000
C01240=76.021,61.028,12.888,-166.7646,-16.1238,0.0000
C01241=78.839,57.492,12.910,-167.3920,-15.6031,0.0000
C01242=80.787,55.140,12.963,-168.0743,-13.2504,0.0000
C01243=82.225,53.620,13.031,-169.6468,-9.9388,0.0000
C01244=83.471,52.459,13.096,-172.2443,-6.9824,0.0000
C01245=84.717,51.269,13.142,-175.1396,-4.9760,0.0000
C01246=86.123,49.643,13.164,-177.4574,-3.2553,0.0000
C01247=87.740,47.377,13.175,-178.9732,-1.5582,0.0000
C01248=89.341,44.743,13.184,-179.7826,-0.3883,0.0000
C01249=90.704,42.074,13.193,-179.9651,-0.0742,0.0000
C01250=91.855,39.526,13.199,-179.9962,-0.0087,0.0000
C01251=92.901,37.002,13.199,-179.9965,-0.0088,0.0000
C01252=93.888,34.387,13.193,-179.9722,-0.0771,0.0000
C01253=94.812,31.535,13.184,-179.8791,-0.4283,0.0000
C01254=95.542,28.540,13.175,-179.6240,-1.8276,0.0000
C01255=96.000,25.795,13.164,-179.4947,-4.0964,0.0000
C01256=96.157,23.652,13.142,-179.9177,-6.9384,0.0000
C01257=96.117,21.929,13.096,179.4441,-10.3652,0.0000
C01258=96.057,20.227,13.031,179.6976,-14.2025,0.0000
C01259=96.115,18.135,12.963,-179.0166,-17.5286,0.0000
C01260=96.401,15.094,12.910,-177.7490,-19.5770,0.0000
C01261=96.908,10.602,12.888,-177.8177,-20.3410,0.0000
C01262=97.322,5.562,12.887,-178.7655,-20.4533,0.0000
C01263=97.482,0.000,12.888,179.9999,-20.4747,0.0000
C01264=97.322,-5.562,12.887,178.7657,-20.4533,0.0000
C01265=96.908,-10.602,12.888,177.8179,-20.3410,0.0000
C01266=96.401,-15.094,12.910,177.7489,-19.5769,0.0000
C01267=96.115,-18.135,12.963,179.0166,-17.5286,0.0000
C01268=96.057,-20.227,13.031,-179.6976,-14.2025,0.0000
C01269=96.117,-21.929,13.096,-179.4441,-10.3652,0.0000
C01270=96.157,-23.652,13.142,179.9177,-6.9384,0.0000
C01271=96.000,-25.795,13.164,179.4947,-4.0964,0.0000
C01272=95.542,-28.540,13.175,179.6240,-1.8276,0.0000
C01273=94.812,-31.535,13.184,179.8791,-0.4283,0.0000
C01274=93.888,-34.387,13.193,179.9722,-0.0771,0.0000
C01275=92.901,-37.002,13.199,179.9965,-0.0088,0.0000
C01276=91.855,-39.526,13.199,179.9962,-0.0087,0.0000
C01277=90.704,-42.074,13.193,179.9651,-0.0742,0.0000
C01278=89.341,-44.743,13.184,179.7826,-0.3883,0.0000
C01279=87.740,-47.377,13.175,178.9732,-1.5582,0.0000
C01280=86.123,-49.643,13.164,177.4574,-3.2553,0.0000
C01281=84.717,-51.269,13.142,175.1396,-4.9760,0.0000
C01282=83.471,-52.459,13.096,172.2443,-6.9824,0.0000
C01283=82.225,-53.620,13.031,169.6468,-9.9388,0.0000
C01284=80.787,-55.140,12.963,168.0743,-13.2504,0.0000
C01285=78.839,-57.492,12.910,167.3919,-15.6031,0.0000
C01286=76.021,-61.028,12.888,166.7648,-16.1239,0.0000
C01287=72.750,-64.884,12.887,166.0456,-15.5868,0.0000
C01288=68.930,-68.930,12.888,165.2101,-14.7897,0.0000
C01289=64.884,-72.750,12.887,164.4133,-13.9544,0.0000
C01290=61.028,-76.021,12.888,163.8762,-13.2354,0.0000
C01291=57.492,-78.839,12.910,164.3969,-12.6080,0.0000
C01292=55.140,-80.787,12.963,166.7496,-11.9257,0.0000
C01293=53.620,-82.225,13.031,170.0612,-10.3532,0.0000
C01294=52.459,-83.471,13.096,173.0176,-7.7557,0.0000
C01295=51.269,-84.717,13.142,175.0240,-4.8604,0.0000
C01296=49.643,-86.123,13.164,176.7447,-2.5426,0.0000
C01297=47.377,-87.740,13.175,178.4418,-1.0268,0.0000
C01298=44.743,-89.341,13.184,179.6117,-0.2174,0.0000
C01299=42.074,-90.704,13.193,179.9258,-0.0349,0.0000
C01300=39.526,-91.855,13.199,179.9913,-0.0038,0.0000
C01301=37.002,-92.901,13.199,179.9912,-0.0035,0.0000
C01302=34.387,-93.888,13.193,179.9229,-0.0278,0.0000
C01303=31.535,-94.812,13.184,179.5717,-0.1209,0.0000
C01304=28.540,-95.542,13.175,178.1724,-0.3760,0.0000
C01305=25.795,-96.000,13.164,175.9036,-0.5053,0.0000
C01306=23.652,-96.157,13.142,173.0616,-0.0823,0.0000
C01307=21.929,-96.117,13.096,169.6348,0.5559,0.0000
C01308=20.227,-96.057,13.031,165.7975,0.3024,0.0000
C01309=18.135,-96.115,12.963,162.4714,-0.9834,0.0000
C01310=15.094,-96.401,12.910,160.4230,-2.2510,0.0000
C01311=10.602,-96.908,12.888,159.6590,-2.1823,0.0000
C01312=5.562,-97.322,12.887,159.5467,-1.2345,0.0000
C01313=0.000,-97.482,12.888,159.5253,0.0001,0.0000
C01314=0.000,-97.482,12.888,159.5253,0.0001,0.0000
C01315=-5.562,-97.322,12.887,159.5467,1.2343,0.0000
C01316=-10.602,-96.908,12.888,159.6590,2.1821,0.0000
C01317=-15.094,-96.401,12.910,160.4231,2.2511,0.0000
C01318=-18.135,-96.115,12.963,162.4714,0.9834,0.0000
C01319=-20.227,-96.057,13.031,165.7975,-0.3024,0.0000
C01320=-21.929,-96.117,13.096,169.6348,-0.5559,0.0000
C01321=-23.652,-96.157,13.142,173.0616,0.0823,0.0000
C01322=-25.795,-96.000,13.164,175.9036,0.5053,0.0000
C01323=-28.540,-95.542,13.175,178.1724,0.3760,0.0000
C01324=-31.535,-94.812,13.184,179.5717,0.1209,0.0000
C01325=-34.387,-93.888,13.193,179.9229,0.0278,0.0000
C01326=-37.002,-92.901,13.199,179.9912,0.0035,0.0000
C01327=-39.526,-91.855,13.199,179.9913,0.0038,0.0000
C01328=-42.074,-90.704,13.193,179.9258,0.0349,0.0000
C01329=-44.743,-89.341,13.184,179.6117,0.2174,0.0000
C01330=-47.377,-87.740,13.175,178.4418,1.0268,0.0000
C01331=-49.643,-86.123,13.164,176.7447,2.5426,0.0000
C01332=-51.269,-84.717,13.142,175.0240,4.8604,0.0000
C01333=-52.459,-83.471,13.096,173.0176,7.7557,0.0000
C01334=-53.620,-82.225,13.031,170.0612,10.3532,0.0000
C01335=-55.140,-80.787,12.963,166.7496,11.9257,0.0000
C01336=-57.492,-78.839,12.910,164.3969,12.6081,0.0000
C01337=-61.028,-76.021,12.888,163.8761,13.2352,0.0000
C01338=-64.884,-72.750,12.887,164.4132,13.9544,0.0000
C01339=-68.930,-68.930,12.888,165.2103,14.7899,0.0000
C01340=-72.750,-64.884,12.887,166.0456,15.5867,0.0000
C01341=-76.021,-61.028,12.888,166.7646,16.1238,0.0000
C01342=-78.839,-57.492,12.910,167.3920,15.6031,0.0000
C01343=-80.787,-55.140,12.963,168.0743,13.2504,0.0000
C01344=-82.225,-53.620,13.031,169.6468,9.9388,0.0000
C01345=-83.471,-52.459,13.096,172.2443,6.9824,0.0000
C01346=-84.717,-51.269,13.142,175.1396,4.9760,0.0000
C01347=-86.123,-49.643,13.164,177.4574,3.2553,0.0000
C01348=-87.740,-47.377,13.175,178.9732,1.5582,0.0000
C01349=-89.341,-44.743,13.184,179.7826,0.3883,0.0000
C01350=-90.704,-42.074,13.193,179.9651,0.0742,0.0000
C01351=-91.855,-39.526,13.199,179.9962,0.0087,0.0000
C01352=-92.901,-37.002,13.199,179.9965,0.0088,0.0000
C01353=-93.888,-34.387,13.193,179.9722,0.0771,0.0000
C01354=-94.812,-31.535,13.184,179.8791,0.4283,0.0000
C01355=-95.542,-28.540,13.175,179.6240,1.8276,0.0000
C01356=-96.000,-25.795,13.164,179.4947,4.0964,0.0000
C01357=-96.157,-23.652,13.142,179.9177,6.9384,0.0000
C01358=-96.117,-21.929,13.096,-179.4441,10.3652,0.0000
C01359=-96.057,-20.227,13.031,-179.6976,14.2025,0.0000
C01360=-96.115,-18.135,12.963,179.0166,17.5286,0.0000
C01361=-96.401,-15.094,12.910,177.7490,19.5770,0.0000
C01362=-96.908,-10.602,12.888,177.8177,20.3410,0.0000
C01363=-97.322,-5.562,12.887,178.7655,20.4533,0.0000
C01364=-97.482,0.000,12.888,-179.9999,20.4747,0.0000
C01365=-97.322,5.562,12.887,-178.7657,20.4533,0.0000
C01366=-96.908,10.602,12.888,-177.8179,20.3410,0.0000
C01367=-96.401,15.094,12.910,-177.7489,19.5769,0.0000
C01368=-96.115,18.135,12.963,-179.0166,17.5286,0.0000
C01369=-96.057,20.227,13.031,179.6976,14.2025,0.0000
C01370=-96.117,21.929,13.096,179.4441,10.3652,0.0000
C01371=-96.157,23.652,13.142,-179.9177,6.9384,0.0000
C01372=-96.000,25.795,13.164,-179.4947,4.0964,0.0000
C01373=-95.542,28.540,13.175,-179.6240,1.8276,0.0000
C01374=-94.812,31.535,13.184,-179.8791,0.4283,0.0000
C01375=-93.888,34.387,13.193,-179.9722,0.0771,0.0000
C01376=-92.901,37.002,13.199,-179.9965,0.0088,0.0000
C01377=-91.855,39.526,13.199,-179.9962,0.0087,0.0000
C01378=-90.704,42.074,13.193,-179.9651,0.0742,0.0000
C01379=-89.341,44.743,13.184,-179.7826,0.3883,0.0000
C01380=-87.740,47.377,13.175,-178.9732,1.5582,0.0000
C01381=-86.123,49.643,13.164,-177.4574,3.2553,0.0000
C01382=-84.717,51.269,13.142,-175.1396,4.9760,0.0000
C01383=-83.471,52.459,13.096,-172.2443,6.9824,0.0000
C01384=-82.225,53.620,13.031,-169.6468,9.9388,0.0000
C01385=-80.787,55.140,12.963,-168.0743,13.2504,0.0000
C01386=-78.839,57.492,12.910,-167.3919,15.6031,0.0000
C01387=-76.021,61.028,12.888,-166.7648,16.1239,0.0000
C01388=-72.750,64.884,12.887,-166.0456,15.5868,0.0000
C01389=-68.930,68.930,12.888,-165.2101,14.7897,0.0000
C01390=-64.884,72.750,12.887,-164.4133,13.9544,0.0000
C01391=-61.028,76.021,12.888,-163.8762,13.2354,0.0000
C01392=-57.492,78.839,12.910,-164.3969,12.6080,0.0000
C01393=-55.140,80.787,12.963,-166.7496,11.9257,0.0000
C01394=-53.620,82.225,13.031,-170.0612,10.3532,0.0000
C01395=-52.459,83.471,13.096,-173.0176,7.7557,0.0000
C01396=-51.269,84.717,13.142,-175.0240,4.8604,0.0000
C01397=-49.643,86.123,13.164,-176.7447,2.5426,0.0000
C01398=-47.377,87.740,13.175,-178.4418,1.0268,0.0000
C01399=-44.743,89.341,13.184,-179.6117,0.2174,0.0000
C01400=-42.074,90.704,13.193,-179.9258,0.0349,0.0000
C01401=-39.526,91.855,13.199,-179.9913,0.0038,0.0000
C01402=-37.002,92.901,13.199,-179.9912,0.0035,0.0000
C01403=-34.387,93.888,13.193,-179.9229,0.0278,0.0000
C01404=-31.535,94.812,13.184,-179.5717,0.1209,0.0000
C01405=-28.540,95.542,13.175,-178.1724,0.3760,0.0000
C01406=-25.795,96.000,13.164,-175.9036,0.5053,0.0000
C01407=-23.652,96.157,13.142,-173.0616,0.0823,0.0000
C01408=-21.929,96.117,13.096,-169.6348,-0.5559,0.0000
C01409=-20.227,96.057,13.031,-165.7975,-0.3024,0.0000
C01410=-18.135,96.115,12.963,-162.4714,0.9834,0.0000
C01411=-15.094,96.401,12.910,-160.4231,2.2511,0.0000
C01412=-10.602,96.908,12.888,-159.6590,2.1821,0.0000
C01413=-5.562,97.322,12.887,-159.5467,1.2343,0.0000
C01414=0.000,97.482,12.888,-159.5253,0.0001,0.0000
C01415=0.000,96.668,14.931,-157.0799,0.0002,0.0000
C01416=5.488,96.511,14.930,-157.1034,-1.3945,0.0000
C01417=10.476,96.104,14.932,-157.2237,-2.4088,0.0000
C01418=14.942,95.628,14.964,-158.0572,-2.1867,0.0000
C01419=17.951,95.422,15.043,-160.4780,-0.1533,0.0000
C01420=20.020,95.481,15.144,-164.5717,1.5921,0.0000
C01421=21.708,95.685,15.242,-169.0703,1.6612,0.0000
C01422=23.417,95.878,15.312,-172.7054,0.5194,0.0000
C01423=25.541,95.862,15.345,-175.6685,-0.3095,0.0000
C01424=28.302,95.513,15.362,-178.1073,-0.3286,0.0000
C01425=31.347,94.846,15.376,-179.5951,-0.1072,0.0000
C01426=34.268,93.927,15.390,-179.9213,-0.0281,0.0000
C01427=36.962,92.916,15.399,-179.9911,-0.0035,0.0000
C01428=39.566,91.838,15.399,-179.9913,-0.0038,0.0000
C01429=42.186,90.648,15.390,-179.9245,-0.0358,0.0000
C01430=44.901,89.232,15.376,-179.6379,-0.2105,0.0000
C01431=47.525,87.551,15.362,-178.4292,-1.1064,0.0000
C01432=49.724,85.845,15.345,-176.7161,-2.8475,0.0000
C01433=51.237,84.354,15.312,-175.1925,-5.5361,0.0000
C01434=52.309,83.010,15.242,-173.3810,-8.9256,0.0000
C01435=53.359,81.672,15.144,-170.0464,-12.1229,0.0000
C01436=54.780,80.167,15.043,-165.8238,-13.9722,0.0000
C01437=57.054,78.185,14.964,-162.6789,-14.4598,0.0000
C01438=60.548,75.364,14.932,-161.9108,-14.9574,0.0000
C01439=64.363,72.124,14.930,-162.4709,-15.7183,0.0000
C01440=68.355,68.355,14.931,-163.3542,-16.6460,0.0000
C01441=72.124,64.363,14.930,-164.2816,-17.5289,0.0000
C01442=75.364,60.548,14.932,-165.0425,-18.0890,0.0000
C01443=78.185,57.054,14.964,-165.5404,-17.3211,0.0000
C01444=80.167,54.780,15.043,-166.0278,-14.1762,0.0000
C01445=81.672,53.359,15.144,-167.8771,-9.9536,0.0000
C01446=83.010,52.309,15.242,-171.0744,-6.6190,0.0000
C01447=84.354,51.237,15.312,-174.4639,-4.8075,0.0000
C01448=85.845,49.724,15.345,-177.1525,-3.2839,0.0000
C01449=87.551,47.525,15.362,-178.8936,-1.5708,0.0000
C01450=89.232,44.901,15.376,-179.7895,-0.3621,0.0000
C01451=90.648,42.186,15.390,-179.9642,-0.0755,0.0000
C01452=91.838,39.566,15.399,-179.9962,-0.0087,0.0000
C01453=92.916,36.962,15.399,-179.9965,-0.0089,0.0000
C01454=93.927,34.268,15.390,-179.9719,-0.0787,0.0000
C01455=94.846,31.347,15.376,-179.8928,-0.4049,0.0000
C01456=95.513,28.302,15.362,-179.6714,-1.8927,0.0000
C01457=95.862,25.541,15.345,-179.6905,-4.3315,0.0000
C01458=95.878,23.417,15.312,179.4806,-7.2946,0.0000
C01459=95.685,21.708,15.242,178.3388,-10.9297,0.0000
C01460=95.481,20.020,15.144,178.4079,-15.4283,0.0000
C01461=95.422,17.951,15.043,-179.8467,-19.5220,0.0000
C01462=95.628,14.942,14.964,-177.8133,-21.9428,0.0000
C01463=96.104,10.476,14.932,-177.5912,-22.7763,0.0000
C01464=96.511,5.488,14.930,-178.6055,-22.8966,0.0000
C01465=96.668,0.000,14.931,179.9998,-22.9201,0.0000
C01466=96.511,-5.488,14.930,178.6057,-22.8966,0.0000
C01467=96.104,-10.476,14.932,177.5915,-22.7763,0.0000
C01468=95.628,-14.942,14.964,177.8131,-21.9428,0.0000
C01469=95.422,-17.951,15.043,179.8467,-19.5220,0.0000
C01470=95.481,-20.020,15.144,-178.4079,-15.4283,0.0000
C01471=95.685,-21.708,15.242,-178.3388,-10.9297,0.0000
C01472=95.878,-23.417,15.312,-179.4806,-7.2946,0.0000
C01473=95.862,-25.541,15.345,179.6905,-4.3315,0.0000
C01474=95.513,-28.302,15.362,179.6714,-1.8927,0.0000
C01475=94.846,-31.347,15.376,179.8928,-0.4049,0.0000
C01476=93.927,-34.268,15.390,179.9719,-0.0787,0.0000
C01477=92.916,-36.962,15.399,179.9965,-0.0089,0.0000
C01478=91.838,-39.566,15.399,179.9962,-0.0087,0.0000
C01479=90.648,-42.186,15.390,179.9642,-0.0755,0.0000
C01480=89.232,-44.901,15.376,179.7895,-0.3621,0.0000
C01481=87.551,-47.525,15.362,178.8936,-1.5708,0.0000
C01482=85.845,-49.724,15.345,177.1525,-3.2839,0.0000
C01483=84.354,-51.237,15.312,174.4639,-4.8075,0.0000
C01484=83.010,-52.309,15.242,171.0744,-6.6190,0.0000
C01485=81.672,-53.359,15.144,167.8771,-9.9536,0.0000
C01486=80.167,-54.780,15.043,166.0278,-14.1762,0.0000
C01487=78.185,-57.054,14.964,165.5402,-17.3211,0.0000
C01488=75.364,-60.548,14.932,165.0426,-18.0892,0.0000
C01489=72.124,-64.363,14.930,164.2817,-17.5291,0.0000
C01490=68.355,-68.355,14.931,163.3540,-16.6458,0.0000
C01491=64.363,-72.124,14.930,162.4711,-15.7184,0.0000
C01492=60.548,-75.364,14.932,161.9110,-14.9575,0.0000
C01493=57.054,-78.185,14.964,162.6789,-14.4596,0.0000
C01494=54.780,-80.167,15.043,165.8238,-13.9722,0.0000
C01495=53.359,-81.672,15.144,170.0464,-12.1229,0.0000
C01496=52.309,-83.010,15.242,173.3810,-8.9256,0.0000
C01497=51.237,-84.354,15.312,175.1925,-5.5361,0.0000
C01498=49.724,-85.845,15.345,176.7161,-2.8475,0.0000
C01499=47.525,-87.551,15.362,178.4292,-1.1064,0.0000
C01500=44.901,-89.232,15.376,179.6379,-0.2105,0.0000
C01501=42.186,-90.648,15.390,179.9245,-0.0358,0.0000
C01502=39.566,-91.838,15.399,179.9913,-0.0038,0.0000
C01503=36.962,-92.916,15.399,179.9911,-0.0035,0.0000
C01504=34.268,-93.927,15.390,179.9213,-0.0281,0.0000
C01505=31.347,-94.846,15.376,179.5951,-0.1072,0.0000
C01506=28.302,-95.513,15.362,178.1073,-0.3286,0.0000
C01507=25.541,-95.862,15.345,175.6685,-0.3095,0.0000
C01508=23.417,-95.878,15.312,172.7054,0.5194,0.0000
C01509=21.708,-95.685,15.242,169.0703,1.6612,0.0000
C01510=20.020,-95.481,15.144,164.5717,1.5921,0.0000
C01511=17.951,-95.422,15.043,160.4780,-0.1533,0.0000
C01512=14.942,-95.628,14.964,158.0572,-2.1867,0.0000
C01513=10.476,-96.104,14.932,157.2237,-2.4088,0.0000
C01514=5.488,-96.511,14.930,157.1034,-1.3945,0.0000
C01515=0.000,-96.668,14.931,157.0799,0.0002,0.0000
C01516=0.000,-96.668,14.931,157.0799,0.0002,0.0000
C01517=-5.488,-96.511,14.930,157.1034,1.3943,0.0000
C01518=-10.476,-96.104,14.932,157.2237,2.4085,0.0000
C01519=-14.942,-95.628,14.964,158.0572,2.1869,0.0000
C01520=-17.951,-95.422,15.043,160.4780,0.1533,0.0000
C01521=-20.020,-95.481,15.144,164.5717,-1.5921,0.0000
C01522=-21.708,-95.685,15.242,169.0703,-1.6612,0.0000
C01523=-23.417,-95.878,15.312,172.7054,-0.5194,0.0000
C01524=-25.541,-95.862,15.345,175.6685,0.3095,0.0000
C01525=-28.302,-95.513,15.362,178.1073,0.3286,0.0000
C01526=-31.347,-94.846,15.376,179.5951,0.1072,0.0000
C01527=-34.268,-93.927,15.390,179.9213,0.0281,0.0000
C01528=-36.962,-92.916,15.399,179.9911,0.0035,0.0000
C01529=-39.566,-91.838,15.399,179.9913,0.0038,0.0000
C01530=-42.186,-90.648,15.390,179.9245,0.0358,0.0000
C01531=-44.901,-89.232,15.376,179.6379,0.2105,0.0000
C01532=-47.525,-87.551,15.362,178.4292,1.1064,0.0000
C01533=-49.724,-85.845,15.345,176.7161,2.8475,0.0000
C01534=-51.237,-84.354,15.312,175.1925,5.5361,0.0000
C01535=-52.309,-83.010,15.242,173.3810,8.9256,0.0000
C01536=-53.359,-81.672,15.144,170.0464,12.1229,0.0000
C01537=-54.780,-80.167,15.043,165.8238,13.9722,0.0000
C01538=-57.054,-78.185,14.964,162.6789,14.4598,0.0000
C01539=-60.548,-75.364,14.932,161.9108,14.9574,0.0000
C01540=-64.363,-72.124,14.930,162.4709,15.7183,0.0000
C01541=-68.355,-68.355,14.931,163.3542,16.6460,0.0000
C01542=-72.124,-64.363,14.930,164.2816,17.5289,0.0000
C01543=-75.364,-60.548,14.932,165.0425,18.0890,0.0000
C01544=-78.185,-57.054,14.964,165.5404,17.3211,0.0000
C01545=-80.167,-54.780,15.043,166.0278,14.1762,0.0000
C01546=-81.672,-53.359,15.144,167.8771,9.9536,0.0000
C01547=-83.010,-52.309,15.242,171.0744,6.6190,0.0000
C01548=-84.354,-51.237,15.312,174.4639,4.8075,0.0000
C01549=-85.845,-49.724,15.345,177.1525,3.2839,0.0000
C01550=-87.551,-47.525,15.362,178.8936,1.5708,0.0000
C01551=-89.232,-44.901,15.376,179.7895,0.3621,0.0000
C01552=-90.648,-42.186,15.390,179.9642,0.0755,0.0000
C01553=-91.838,-39.566,15.399,179.9962,0.0087,0.0000
C01554=-92.916,-36.962,15.399,179.9965,0.0089,0.0000
C01555=-93.927,-34.268,15.390,179.9719,0.0787,0.0000
C01556=-94.846,-31.347,15.376,179.8928,0.4049,0.0000
C01557=-95.513,-28.302,15.362,179.6714,1.8927,0.0000
C01558=-95.862,-25.541,15.345,179.6905,4.3315,0.0000
C01559=-95.878,-23.417,15.312,-179.4806,7.2946,0.0000
C01560=-95.685,-21.708,15.242,-178.3388,10.9297,0.0000
C01561=-95.481,-20.020,15.144,-178.4079,15.4283,0.0000
C01562=-95.422,-17.951,15.043,179.8467,19.5220,0.0000
C01563=-95.628,-14.942,14.964,177.8133,21.9428,0.0000
C01564=-96.104,-10.476,14.932,177.5912,22.7763,0.0000
C01565=-96.511,-5.488,14.930,178.6055,22.8966,0.0000
C01566=-96.668,0.000,14.931,-179.9998,22.9201,0.0000
C01567=-96.511,5.488,14.930,-178.6057,22.8966,0.0000
C01568=-96.104,10.476,14.932,-177.5915,22.7763,0.0000
C01569=-95.628,14.942,14.964,-177.8131,21.9428,0.0000
C01570=-95.422,17.951,15.043,-179.8467,19.5220,0.0000
C01571=-95.481,20.020,15.144,178.4079,15.4283,0.0000
C01572=-95.685,21.708,15.242,178.3388,10.9297,0.0000
C01573=-95.878,23.417,15.312,179.4806,7.2946,0.0000
C01574=-95.862,25.541,15.345,-179.6905,4.3315,0.0000
C01575=-95.513,28.302,15.362,-179.6714,1.8927,0.0000
C01576=-94.846,31.347,15.376,-179.8928,0.4049,0.0000
C01577=-93.927,34.268,15.390,-179.9719,0.0787,0.0000
C01578=-92.916,36.962,15.399,-179.9965,0.0089,0.0000
C01579=-91.838,39.566,15.399,-179.9962,0.0087,0.0000
C01580=-90.648,42.186,15.390,-179.9642,0.0755,0.0000
C01581=-89.232,44.901,15.376,-179.7895,0.3621,0.0000
C01582=-87.551,47.525,15.362,-178.8936,1.5708,0.0000
C01583=-85.845,49.724,15.345,-177.1525,3.2839,0.0000
C01584=-84.354,51.237,15.312,-174.4639,4.8075,0.0000
C01585=-83.010,52.309,15.242,-171.0744,6.6190,0.0000
C01586=-81.672,53.359,15.144,-167.8771,9.9536,0.0000
C01587=-80.167,54.780,15.043,-166.0278,14.1762,0.0000
C01588=-78.185,57.054,14.964,-165.5402,17.3211,0.0000
C01589=-75.364,60.548,14.932,-165.0426,18.0892,0.0000
C01590=-72.124,64.363,14.930,-164.2817,17.5291,0.0000
C01591=-68.355,68.355,14.931,-163.3540,16.6458,0.0000
C01592=-64.363,72.124,14.930,-162.4711,15.7184,0.0000
C01593=-60.548,75.364,14.932,-161.9110,14.9575,0.0000
C01594=-57.054,78.185,14.964,-162.6789,14.4596,0.0000
C01595=-54.780,80.167,15.043,-165.8238,13.9722,0.0000
C01596=-53.359,81.672,15.144,-170.0464,12.1229,0.0000
C01597=-52.309,83.010,15.242,-173.3810,8.9256,0.0000
C01598=-51.237,84.354,15.312,-175.1925,5.5361,0.0000
C01599=-49.724,85.845,15.345,-176.7161,2.8475,0.0000
C01600=-47.525,87.551,15.362,-178.4292,1.1064,0.0000
C01601=-44.901,89.232,15.376,-179.6379,0.2105,0.0000
C01602=-42.186,90.648,15.390,-179.9245,0.0358,0.0000
C01603=-39.566,91.838,15.399,-179.9913,0.0038,0.0000
C01604=-36.962,92.916,15.399,-179.9911,0.0035,0.0000
C01605=-34.268,93.927,15.390,-179.9213,0.0281,0.0000
C01606=-31.347,94.846,15.376,-179.5951,0.1072,0.0000
C01607=-28.302,95.513,15.362,-178.1073,0.3286,0.0000
C01608=-25.541,95.862,15.345,-175.6685,0.3095,0.0000
C01609=-23.417,95.878,15.312,-172.7054,-0.5194,0.0000
C01610=-21.708,95.685,15.242,-169.0703,-1.6612,0.0000
C01611=-20.020,95.481,15.144,-164.5717,-1.5921,0.0000
C01612=-17.951,95.422,15.043,-160.4780,0.1533,0.0000
C01613=-14.942,95.628,14.964,-158.0572,2.1869,0.0000
C01614=-10.476,96.104,14.932,-157.2237,2.4085,0.0000
C01615=-5.488,96.511,14.930,-157.1034,1.3943,0.0000
C01616=0.000,96.668,14.931,-157.0799,0.0002,0.0000
C01617=0.000,95.772,16.941,-154.8859,0.0002,0.0000
C01618=5.406,95.617,16.939,-154.9111,-1.5415,0.0000
C01619=10.339,95.219,16.941,-155.0372,-2.5925,0.0000
C01620=14.774,94.777,16.986,-155.9394,-1.9734,0.0000
C01621=17.748,94.656,17.095,-158.8449,1.0095,0.0000
C01622=19.790,94.842,17.237,-163.9074,3.1515,0.0000
C01623=21.462,95.203,17.374,-169.0788,2.8690,0.0000
C01624=23.155,95.565,17.473,-172.7347,1.2030,0.0000
C01625=25.257,95.708,17.521,-175.6219,-0.0566,0.0000
C01626=28.035,95.481,17.545,-178.1277,-0.2593,0.0000
C01627=31.135,94.884,17.565,-179.6493,-0.0862,0.0000
C01628=34.135,93.972,17.585,-179.9232,-0.0272,0.0000
C01629=36.917,92.934,17.598,-179.9915,-0.0033,0.0000
C01630=39.610,91.818,17.598,-179.9916,-0.0037,0.0000
C01631=42.311,90.585,17.585,-179.9265,-0.0351,0.0000
C01632=45.077,89.109,17.565,-179.6910,-0.1870,0.0000
C01633=47.692,87.339,17.545,-178.4926,-1.1409,0.0000
C01634=49.816,85.535,17.521,-176.8613,-3.0589,0.0000
C01635=51.202,83.948,17.473,-175.6939,-5.9938,0.0000
C01636=52.143,82.495,17.374,-174.2326,-9.7525,0.0000
C01637=53.070,81.058,17.237,-170.6271,-13.6544,0.0000
C01638=54.382,79.482,17.095,-165.3630,-15.9654,0.0000
C01639=56.571,77.464,16.986,-161.2176,-16.2439,0.0000
C01640=60.019,74.640,16.941,-160.1409,-16.5495,0.0000
C01641=63.789,71.434,16.939,-160.7051,-17.3299,0.0000
C01642=67.721,67.721,16.941,-161.6626,-18.3377,0.0000
C01643=71.434,63.789,16.939,-162.6700,-19.2947,0.0000
C01644=74.640,60.019,16.941,-163.4503,-19.8589,0.0000
C01645=77.464,56.571,16.986,-163.7563,-18.7825,0.0000
C01646=79.482,54.382,17.095,-164.0346,-14.6370,0.0000
C01647=81.058,53.070,17.237,-166.3456,-9.3729,0.0000
C01648=82.495,52.143,17.374,-170.2475,-5.7674,0.0000
C01649=83.948,51.202,17.473,-174.0062,-4.3061,0.0000
C01650=85.535,49.816,17.521,-176.9411,-3.1387,0.0000
C01651=87.339,47.692,17.545,-178.8591,-1.5074,0.0000
C01652=89.109,45.077,17.565,-179.8130,-0.3090,0.0000
C01653=90.585,42.311,17.585,-179.9649,-0.0735,0.0000
C01654=91.818,39.610,17.598,-179.9963,-0.0084,0.0000
C01655=92.934,36.917,17.598,-179.9967,-0.0085,0.0000
C01656=93.972,34.135,17.585,-179.9728,-0.0768,0.0000
C01657=94.884,31.135,17.565,-179.9138,-0.3507,0.0000
C01658=95.481,28.035,17.545,-179.7407,-1.8723,0.0000
C01659=95.708,25.257,17.521,-179.9434,-4.3781,0.0000
C01660=95.565,23.155,17.473,178.7970,-7.2653,0.0000
C01661=95.203,21.462,17.374,177.1310,-10.9212,0.0000
C01662=94.842,19.790,17.237,176.8485,-16.0926,0.0000
C01663=94.656,17.748,17.095,178.9905,-21.1551,0.0000
C01664=94.777,14.774,16.986,-178.0266,-24.0606,0.0000
C01665=95.219,10.339,16.941,-177.4075,-24.9628,0.0000
C01666=95.617,5.406,16.939,-178.4585,-25.0889,0.0000
C01667=95.772,0.000,16.941,179.9998,-25.1141,0.0000
C01668=95.617,-5.406,16.939,178.4588,-25.0889,0.0000
C01669=95.219,-10.339,16.941,177.4079,-24.9628,0.0000
C01670=94.777,-14.774,16.986,178.0264,-24.0606,0.0000
C01671=94.656,-17.748,17.095,-178.9905,-21.1551,0.0000
C01672=94.842,-19.790,17.237,-176.8485,-16.0926,0.0000
C01673=95.203,-21.462,17.374,-177.1310,-10.9212,0.0000
C01674=95.565,-23.155,17.473,-178.7970,-7.2653,0.0000
C01675=95.708,-25.257,17.521,179.9434,-4.3781,0.0000
C01676=95.481,-28.035,17.545,179.7407,-1.8723,0.0000
C01677=94.884,-31.135,17.565,179.9138,-0.3507,0.0000
C01678=93.972,-34.135,17.585,179.9728,-0.0768,0.0000
C01679=92.934,-36.917,17.598,179.9967,-0.0085,0.0000
C01680=91.818,-39.610,17.598,179.9963,-0.0084,0.0000
C01681=90.585,-42.311,17.585,179.9649,-0.0735,0.0000
C01682=89.109,-45.077,17.565,179.8130,-0.3090,0.0000
C01683=87.339,-47.692,17.545,178.8591,-1.5074,0.0000
C01684=85.535,-49.816,17.521,176.9411,-3.1387,0.0000
C01685=83.948,-51.202,17.473,174.0062,-4.3061,0.0000
C01686=82.495,-52.143,17.374,170.2475,-5.7674,0.0000
C01687=81.058,-53.070,17.237,166.3456,-9.3729,0.0000
C01688=79.482,-54.382,17.095,164.0346,-14.6370,0.0000
C01689=77.464,-56.571,16.986,163.7561,-18.7824,0.0000
C01690=74.640,-60.019,16.941,163.4505,-19.8591,0.0000
C01691=71.434,-63.789,16.939,162.6701,-19.2949,0.0000
C01692=67.721,-67.721,16.941,161.6623,-18.3374,0.0000
C01693=63.789,-71.434,16.939,160.7053,-17.3300,0.0000
C01694=60.019,-74.640,16.941,160.1411,-16.5497,0.0000
C01695=56.571,-77.464,16.986,161.2175,-16.2437,0.0000
C01696=54.382,-79.482,17.095,165.3630,-15.9654,0.0000
C01697=53.070,-81.058,17.237,170.6271,-13.6544,0.0000
C01698=52.143,-82.495,17.374,174.2326,-9.7525,0.0000
C01699=51.202,-83.948,17.473,175.6939,-5.9938,0.0000
C01700=49.816,-85.535,17.521,176.8613,-3.0589,0.0000
C01701=47.692,-87.339,17.545,178.4926,-1.1409,0.0000
C01702=45.077,-89.109,17.565,179.6910,-0.1870,0.0000
C01703=42.311,-90.585,17.585,179.9265,-0.0351,0.0000
C01704=39.610,-91.818,17.598,179.9916,-0.0037,0.0000
C01705=36.917,-92.934,17.598,179.9915,-0.0033,0.0000
C01706=34.135,-93.972,17.585,179.9232,-0.0272,0.0000
C01707=31.135,-94.884,17.565,179.6493,-0.0862,0.0000
C01708=28.035,-95.481,17.545,178.1277,-0.2593,0.0000
C01709=25.257,-95.708,17.521,175.6219,-0.0566,0.0000
C01710=23.155,-95.565,17.473,172.7347,1.2030,0.0000
C01711=21.462,-95.203,17.374,169.0788,2.8690,0.0000
C01712=19.790,-94.842,17.237,163.9074,3.1515,0.0000
C01713=17.748,-94.656,17.095,158.8449,1.0095,0.0000
C01714=14.774,-94.777,16.986,155.9394,-1.9734,0.0000
C01715=10.339,-95.219,16.941,155.0372,-2.5925,0.0000
C01716=5.406,-95.617,16.939,154.9111,-1.5415,0.0000
C01717=0.000,-95.772,16.941,154.8859,0.0002,0.0000
C01718=0.000,-95.772,16.941,154.8859,0.0002,0.0000
C01719=-5.406,-95.617,16.939,154.9111,1.5412,0.0000
C01720=-10.339,-95.219,16.941,155.0372,2.5921,0.0000
C01721=-14.774,-94.777,16.986,155.9394,1.9736,0.0000
C01722=-17.748,-94.656,17.095,158.8449,-1.0095,0.0000
C01723=-19.790,-94.842,17.237,163.9074,-3.1515,0.0000
C01724=-21.462,-95.203,17.374,169.0788,-2.8690,0.0000
C01725=-23.155,-95.565,17.473,172.7347,-1.2030,0.0000
C01726=-25.257,-95.708,17.521,175.6219,0.0566,0.0000
C01727=-28.035,-95.481,17.545,178.1277,0.2593,0.0000
C01728=-31.135,-94.884,17.565,179.6493,0.0862,0.0000
C01729=-34.135,-93.972,17.585,179.9232,0.0272,0.0000
C01730=-36.917,-92.934,17.598,179.9915,0.0033,0.0000
C01731=-39.610,-91.818,17.598,179.9916,0.0037,0.0000
C01732=-42.311,-90.585,17.585,179.9265,0.0351,0.0000
C01733=-45.077,-89.109,17.565,179.6910,0.1870,0.0000
C01734=-47.692,-87.339,17.545,178.4926,1.1409,0.0000
C01735=-49.816,-85.535,17.521,176.8613,3.0589,0.0000
C01736=-51.202,-83.948,17.473,175.6939,5.9938,0.0000
C01737=-52.143,-82.495,17.374,174.2326,9.7525,0.0000
C01738=-53.070,-81.058,17.237,170.6271,13.6544,0.0000
C01739=-54.382,-79.482,17.095,165.3630,15.9654,0.0000
C01740=-56.571,-77.464,16.986,161.2176,16.2439,0.0000
C01741=-60.019,-74.640,16.941,160.1409,16.5495,0.0000
C01742=-63.789,-71.434,16.939,160.7051,17.3299,0.0000
C01743=-67.721,-67.721,16.941,161.6626,18.3377,0.0000
C01744=-71.434,-63.789,16.939,162.6700,19.2947,0.0000
C01745=-74.640,-60.019,16.941,163.4503,19.8589,0.0000
C01746=-77.464,-56.571,16.986,163.7563,18.7825,0.0000
C01747=-79.482,-54.382,17.095,164.0346,14.6370,0.0000
C01748=-81.058,-53.070,17.237,166.3456,9.3729,0.0000
C01749=-82.495,-52.143,17.374,170.2475,5.7674,0.0000
C01750=-83.948,-51.202,17.473,174.0062,4.3061,0.0000
C01751=-85.535,-49.816,17.521,176.9411,3.1387,0.0000
C01752=-87.339,-47.692,17.545,178.8591,1.5074,0.0000
C01753=-89.109,-45.077,17.565,179.8130,0.3090,0.0000
C01754=-90.585,-42.311,17.585,179.9649,0.0735,0.0000
C01755=-91.818,-39.610,17.598,179.9963,0.0084,0.0000
C01756=-92.934,-36.917,17.598,179.9967,0.0085,0.0000
C01757=-93.972,-34.135,17.585,179.9728,0.0768,0.0000
C01758=-94.884,-31.135,17.565,179.9138,0.3507,0.0000
C01759=-95.481,-28.035,17.545,179.7407,1.8723,0.0000
C01760=-95.708,-25.257,17.521,179.9434,4.3781,0.0000
C01761=-95.565,-23.155,17.473,-178.7970,7.2653,0.0000
C01762=-95.203,-21.462,17.374,-177.1310,10.9212,0.0000
C01763=-94.842,-19.790,17.237,-176.8485,16.0926,0.0000
C01764=-94.656,-17.748,17.095,-178.9905,21.1551,0.0000
C01765=-94.777,-14.774,16.986,178.0266,24.0606,0.0000
C01766=-95.219,-10.339,16.941,177.4075,24.9628,0.0000
C01767=-95.617,-5.406,16.939,178.4585,25.0889,0.0000
C01768=-95.772,0.000,16.941,-179.9998,25.1141,0.0000
C01769=-95.617,5.406,16.939,-178.4588,25.0889,0.0000
C01770=-95.219,10.339,16.941,-177.4079,24.9628,0.0000
C01771=-94.777,14.774,16.986,-178.0264,24.0606,0.0000
C01772=-94.656,17.748,17.095,178.9905,21.1551,0.0000
C01773=-94.842,19.790,17.237,176.8485,16.0926,0.0000
C01774=-95.203,21.462,17.374,177.1310,10.9212,0.0000
C01775=-95.565,23.155,17.473,178.7970,7.2653,0.0000
C01776=-95.708,25.257,17.521,-179.9434,4.3781,0.0000
C01777=-95.481,28.035,17.545,-179.7407,1.8723,0.0000
C01778=-94.884,31.135,17.565,-179.9138,0.3507,0.0000
C01779=-93.972,34.135,17.585,-179.9728,0.0768,0.0000
C01780=-92.934,36.917,17.598,-179.9967,0.0085,0.0000
C01781=-91.818,39.610,17.598,-179.9963,0.0084,0.0000
C01782=-90.585,42.311,17.585,-179.9649,0.0735,0.0000
C01783=-89.109,45.077,17.565,-179.8130,0.3090,0.0000
C01784=-87.339,47.692,17.545,-178.8591,1.5074,0.0000
C01785=-85.535,49.816,17.521,-176.9411,3.1387,0.0000
C01786=-83.948,51.202,17.473,-174.0062,4.3061,0.0000
C01787=-82.495,52.143,17.374,-170.2475,5.7674,0.0000
C01788=-81.058,53.070,17.237,-166.3456,9.3729,0.0000
C01789=-79.482,54.382,17.095,-164.0346,14.6370,0.0000
C01790=-77.464,56.571,16.986,-163.7561,18.7824,0.0000
C01791=-74.640,60.019,16.941,-163.4505,19.8591,0.0000
C01792=-71.434,63.789,16.939,-162.6701,19.2949,0.0000
C01793=-67.721,67.721,16.941,-161.6623,18.3374,0.0000
C01794=-63.789,71.434,16.939,-160.7053,17.3300,0.0000
C01795=-60.019,74.640,16.941,-160.1411,16.5497,0.0000
C01796=-56.571,77.464,16.986,-161.2175,16.2437,0.0000
C01797=-54.382,79.482,17.095,-165.3630,15.9654,0.0000
C01798=-53.070,81.058,17.237,-170.6271,13.6544,0.0000
C01799=-52.143,82.495,17.374,-174.2326,9.7525,0.0000
C01800=-51.202,83.948,17.473,-175.6939,5.9938,0.0000
C01801=-49.816,85.535,17.521,-176.8613,3.0589,0.0000
C01802=-47.692,87.339,17.545,-178.4926,1.1409,0.0000
C01803=-45.077,89.109,17.565,-179.6910,0.1870,0.0000
C01804=-42.311,90.585,17.585,-179.9265,0.0351,0.0000
C01805=-39.610,91.818,17.598,-179.9916,0.0037,0.0000
C01806=-36.917,92.934,17.598,-179.9915,0.0033,0.0000
C01807=-34.135,93.972,17.585,-179.9232,0.0272,0.0000
C01808=-31.135,94.884,17.565,-179.6493,0.0862,0.0000
C01809=-28.035,95.481,17.545,-178.1277,0.2593,0.0000
C01810=-25.257,95.708,17.521,-175.6219,0.0566,0.0000
C01811=-23.155,95.565,17.473,-172.7347,-1.2030,0.0000
C01812=-21.462,95.203,17.374,-169.0788,-2.8690,0.0000
C01813=-19.790,94.842,17.237,-163.9074,-3.1515,0.0000
C01814=-17.748,94.656,17.095,-158.8449,-1.0095,0.0000
C01815=-14.774,94.777,16.986,-155.9394,1.9736,0.0000
C01816=-10.339,95.219,16.941,-155.0372,2.5921,0.0000
C01817=-5.406,95.617,16.939,-154.9111,1.5412,0.0000
C01818=0.000,95.772,16.941,-154.8859,0.0002,0.0000
C01819=0.000,94.804,18.916,-152.9230,0.0002,0.0000
C01820=5.317,94.652,18.914,-152.9496,-1.6759,0.0000
C01821=10.190,94.262,18.917,-153.0799,-2.7339,0.0000
C01822=14.592,93.857,18.976,-154.0583,-1.6112,0.0000
C01823=17.528,93.824,19.120,-157.6135,2.4711,0.0000
C01824=19.540,94.146,19.309,-163.8609,4.8105,0.0000
C01825=21.192,94.676,19.493,-169.6633,3.9762,0.0000
C01826=22.867,95.222,19.627,-173.1704,1.8493,0.0000
C01827=24.945,95.538,19.692,-175.7796,0.2187,0.0000
C01828=27.741,95.446,19.726,-178.2343,-0.1783,0.0000
C01829=30.903,94.927,19.753,-179.7329,-0.0604,0.0000
C01830=33.988,94.020,19.780,-179.9280,-0.0252,0.0000
C01831=36.867,92.953,19.798,-179.9922,-0.0031,0.0000
C01832=39.659,91.796,19.798,-179.9923,-0.0034,0.0000
C01833=42.449,90.515,19.780,-179.9313,-0.0331,0.0000
C01834=45.272,88.975,19.753,-179.7684,-0.1462,0.0000
C01835=47.874,87.106,19.726,-178.6253,-1.1228,0.0000
C01836=49.917,85.194,19.692,-177.1673,-3.1412,0.0000
C01837=51.163,83.502,19.627,-176.4604,-6.1368,0.0000
C01838=51.961,81.931,19.493,-175.4363,-10.0997,0.0000
C01839=52.755,80.388,19.309,-171.7434,-14.7955,0.0000
C01840=53.950,78.738,19.120,-165.3862,-17.8366,0.0000
C01841=56.048,76.685,18.976,-160.0047,-17.9574,0.0000
C01842=59.448,73.859,18.917,-158.5544,-18.0188,0.0000
C01843=63.169,70.689,18.914,-159.1051,-18.7977,0.0000
C01844=67.036,67.036,18.916,-160.1259,-19.8744,0.0000
C01845=70.689,63.169,18.914,-161.2021,-20.8947,0.0000
C01846=73.859,59.448,18.917,-161.9809,-21.4453,0.0000
C01847=76.685,56.048,18.976,-162.0428,-19.9955,0.0000
C01848=78.738,53.950,19.120,-162.1634,-14.6138,0.0000
C01849=80.388,52.755,19.309,-165.2045,-8.2566,0.0000
C01850=81.931,51.961,19.493,-169.9003,-4.5637,0.0000
C01851=83.502,51.163,19.627,-173.8632,-3.5396,0.0000
C01852=85.194,49.917,19.692,-176.8588,-2.8327,0.0000
C01853=87.106,47.874,19.726,-178.8772,-1.3747,0.0000
C01854=88.975,45.272,19.753,-179.8538,-0.2316,0.0000
C01855=90.515,42.449,19.780,-179.9669,-0.0687,0.0000
C01856=91.796,39.659,19.798,-179.9966,-0.0077,0.0000
C01857=92.953,36.867,19.798,-179.9969,-0.0078,0.0000
C01858=94.020,33.988,19.780,-179.9748,-0.0720,0.0000
C01859=94.927,30.903,19.753,-179.9396,-0.2671,0.0000
C01860=95.446,27.741,19.726,-179.8217,-1.7657,0.0000
C01861=95.538,24.945,19.692,179.7813,-4.2204,0.0000
C01862=95.222,22.867,19.627,178.1507,-6.8296,0.0000
C01863=94.676,21.192,19.493,176.0238,-10.3367,0.0000
C01864=94.146,19.540,19.309,175.1895,-16.1391,0.0000
C01865=93.824,17.528,19.120,177.5289,-22.3865,0.0000
C01866=93.857,14.592,18.976,-178.3888,-25.9417,0.0000
C01867=94.262,10.190,18.917,-177.2661,-26.9201,0.0000
C01868=94.652,5.317,18.914,-178.3241,-27.0504,0.0000
C01869=94.804,0.000,18.916,179.9998,-27.0770,0.0000
C01870=94.652,-5.317,18.914,178.3244,-27.0504,0.0000
C01871=94.262,-10.190,18.917,177.2665,-26.9201,0.0000
C01872=93.857,-14.592,18.976,178.3885,-25.9416,0.0000
C01873=93.824,-17.528,19.120,-177.5289,-22.3865,0.0000
C01874=94.146,-19.540,19.309,-175.1895,-16.1391,0.0000
C01875=94.676,-21.192,19.493,-176.0238,-10.3367,0.0000
C01876=95.222,-22.867,19.627,-178.1507,-6.8296,0.0000
C01877=95.538,-24.945,19.692,-179.7813,-4.2204,0.0000
C01878=95.446,-27.741,19.726,179.8217,-1.7657,0.0000
C01879=94.927,-30.903,19.753,179.9396,-0.2671,0.0000
C01880=94.020,-33.988,19.780,179.9748,-0.0720,0.0000
C01881=92.953,-36.867,19.798,179.9969,-0.0078,0.0000
C01882=91.796,-39.659,19.798,179.9966,-0.0077,0.0000
C01883=90.515,-42.449,19.780,179.9669,-0.0687,0.0000
C01884=88.975,-45.272,19.753,179.8538,-0.2316,0.0000
C01885=87.106,-47.874,19.726,178.8772,-1.3747,0.0000
C01886=85.194,-49.917,19.692,176.8588,-2.8327,0.0000
C01887=83.502,-51.163,19.627,173.8632,-3.5396,0.0000
C01888=81.931,-51.961,19.493,169.9003,-4.5637,0.0000
C01889=80.388,-52.755,19.309,165.2045,-8.2566,0.0000
C01890=78.738,-53.950,19.120,162.1634,-14.6138,0.0000
C01891=76.685,-56.048,18.976,162.0426,-19.9953,0.0000
C01892=73.859,-59.448,18.917,161.9812,-21.4456,0.0000
C01893=70.689,-63.169,18.914,161.2023,-20.8949,0.0000
